Omron CX-Programmer project NewProject (CX-Programmer 9.74)

# PLC NewPLC1: CJ2M CPU32
I/O table (CPU CJ2M-CPU32): rack 0 slot 0 CJ1W-ID211; rack 0 slot 1 CJ1W-ID211; rack 0 slot 2 CJ1W-OD232; rack 0 slot 3 CJ1W-TC104; rack 0 slot 11 CJ2M-EIP21

## Data types
TYPE s_Steps : STRUCT
  f : INT;  (* Função *)
  p1 : INT;  (* Parametro 1 *)
  p2 : REAL;  (* Parametro 2 *)
END_STRUCT END_TYPE
TYPE s_Estado : STRUCT
  Ciclo : BOOL;  (* Em ciclo produtivo *)
  FimCiclo : BOOL;  (* Finalização ciclo *)
  Estado : BOOL;  (* Estado equipamento *)
  FimTratamento : BOOL;  (* Tratamento Finalizado *)
  OF_Carregada : BOOL;  (* Ordem carregada para máquina *)
  Avaria : BOOL;  (* Máquina em Avaria *)
  Com_OF : BOOL;  (* Máquina com OF carregada *)
  FalhaInjeProd : BOOL;  (* Falta de injeção de produto *)
  FalhaAquecim : BOOL;  (* Falha de aquecimento *)
  AvariaTermicos : BOOL;  (* Avaria de térmicos *)
  TratAbortado : BOOL;  (* Tratamento abortado pelo operador *)
  FalhaEnergia : BOOL;  (* Falha energia *)
  NivelProdBaixo : BOOL;  (* Nível produto químico no depósito baixo *)
  Manual : BOOL;  (* modo manual *)
  Emergencia : BOOL;  (* Paragem Emergência *)
END_STRUCT END_TYPE
TYPE s_of_pss : STRUCT  (* Passo individual do programa a executar *)
  f : INT;  (* Função *)
  p1 : INT;  (* Parametro 1 *)
  p2 : REAL;  (* Parametro 2 *)
  tt : REAL;  (* Totalizador *)
  uni : INT;  (* Unidade do totalizador *)
  rsv : INT Dimensions=[3];
END_STRUCT END_TYPE
TYPE s_pss_exe : STRUCT  (* Passo a executar *)
  pss : s_of_pss;  (* Passo actual a executar *)
  num_pss : INT;  (* Numero do passo actual *)
  ini : BOOL;  (* Inicio - Inicio do passo (Função faz inicializações necessárias) *)
  exe : BOOL;  (* Executar - Condição para funcionar (Função actua se valor igual a 1) *)
  fim : BOOL;  (* Fim - Terminado o passo (Função indica que terminou de executar) *)
  exc : BOOL;  (* Exclusivo - Condição para funções exclusivas (Função exclusiva coloca a 0 ao executar, impedindo que outras o façam) *)
END_STRUCT END_TYPE
TYPE s_trat : STRUCT
  Aspira : BOOL;
  Aquece : BOOL;
  Rotacao : BOOL;
  Injecao : BOOL;
  Ini : BOOL;
  Fim : BOOL;  (* Fim Passo *)
  CicloAtivo : BOOL;
  FimTratamento : BOOL;
END_STRUCT END_TYPE
TYPE s_of : STRUCT
  pss : s_of_pss Dimensions=[12];
END_STRUCT END_TYPE
TYPE s_of_net : STRUCT
  pss : s_Steps Dimensions=[12];
END_STRUCT END_TYPE

## Global symbols (name address type ; comment)
0.00 BOOL  ; Emerg:M1
0.00 BOOL  ; Emergency_M1
0.01 BOOL  ; Bt_start_M1
0.02 BOOL  ; Bt__Stop_M1
0.03 BOOL  ; selector de carga
0.04 BOOL  ; confirma carga
0.05 BOOL  ; Selector Descarga
0.06 BOOL  ; Confirma descarga
0.07 BOOL  ; Sns_flow_M1
0.08 BOOL  ; FC_PRT_M1
0.10 BOOL  ; conf rot M1
0.12 BOOL  ; Mgt_Resist_M1
0.13 BOOL  ; Emergencia
0.14 BOOL  ; bt_start
11.00 BOOL  ; Aux_ro_M1
12.00 BOOL  ; Aux_rot_M2
1.00 BOOL  ; Emerg:M2
1.01 BOOL  ; bt_inicio:M2
1.03 BOOL  ; selector de carga_M2
1.04 BOOL  ; conf carga_M2
1.05 BOOL  ; Sel Desc_M2
1.06 BOOL  ; Conf desc M2
1.07 BOOL  ; Sns_flow_M2
1.08 BOOL  ; FC_PRT_M2
1.10 BOOL  ; conf rot M2
1.12 BOOL  ; MGT_Resist_M2
1.13 BOOL  ; Cmt_Silo_1
1.14 BOOL  ; Cmt_Silo_2
2000 CHANNEL  ; Area_sp_Tc104_M1
2.00 BOOL  ; Girafa
2.01 BOOL  ; Tap_dist-DIR
2.02 BOOL  ; Out_Lig_desv1
2.03 BOOL  ; Out_Desl_desv1
2.04 BOOL  ; out_desv2
2.05 BOOL  ; Out_Desl_desv2
2.06 BOOL  ; Flap_Silo1
2.07 BOOL  ; Flap_Silo2
2.08 BOOL  ; Rotaçao_M1
2.09 BOOL  ; Resist_M1
2.10 BOOL  ; Valv_Aspira_M1
2.11 BOOL  ; Prt_Carga_M1
2.12 BOOL  ; Prt_Desc_M1
2.13 BOOL  ; lmp_auto_m1
2.14 BOOL  ; Lmp_Prt_carga_M1
2.15 BOOL  ; Lmp_Prt_Desc_M1
3.00 BOOL  ; Rotaçao_M2
3.01 BOOL  ; Resist_M2
3.02 BOOL  ; Valv_Aspira_M2
3.03 BOOL  ; Prt_Carga_M2
3.04 BOOL  ; Prt_Desc_M2
3.05 BOOL  ; lmp_auto_m2
3.06 BOOL  ; Lmp_Prt_carga_M2
3.07 BOOL  ; Lmp_Prt_Desc_M2
3.08 BOOL  ; lmp_Start_QE
3.09 BOOL  ; LMP_AVARIA_QE
3.10 BOOL  ; Led_Cmt_desv1
3.11 BOOL  ; Led_Cmt_desv2
3.12 BOOL  ; esquerda
3.13 BOOL  ; Vl_Inver_Tapete
3.14 BOOL  ; Baliza_M7
3.15 BOOL  ; Baliza_M8
C0001 BOOL  ; Cnt_CLC_1
C0002 BOOL  ; Cnt_CLC_2
C0003 BOOL  ; Cnt_CLC_3
C0004 BOOL  ; Cnt_CLC_4
C0005 BOOL  ; Cnt_CLC_5
C0011 BOOL  ; Cnt_CLC_1_M2
C0012 BOOL  ; Cnt_CLC_2_M2
C0013 BOOL  ; T_CLC_3_M2
C0014 BOOL  ; Cnt_CLC_4_M2
C0015 BOOL  ; Cnt_CLC_5_M2
D0 CHANNEL  ; Cntrl_Ns
D15 CHANNEL  ; Str_Msgs_M1
D16 CHANNEL  ; Pop_Inj_M2
D20 CHANNEL  ; T_CLC_1_M2
D21 CHANNEL  ; T_CLC_2
D22 CHANNEL  ; T_CLC_3
D23 CHANNEL  ; T_CLC_4
D24 CHANNEL  ; T_CLC_5
D25 CHANNEL  ; Str_Msgs_M1
D29 CHANNEL  ; Setp_temp_M1
D31 CHANNEL  ; T_CLC_2_M2
D32 CHANNEL  ; T_CLC_3_M2
D33 CHANNEL  ; T_CLC_4_M2
D34 CHANNEL  ; T_CLC_5_M2
D35 CHANNEL  ; Str_Msgs_M2
D38 CHANNEL  ; Area_sp_Tc104_M2
D39 CHANNEL  ; Setp_temp_M2
D5 CHANNEL  ; HMi_Notify
D6 CHANNEL  ; Pop_Inj_M1
D995 CHANNEL  ; Setp_Manual
D999 CHANNEL  ; Setp_Temp_NS
H0.00 BOOL  ; Auto_M1
H0.00 BOOL  ; Auto_M1
H0.08 BOOL  ; ALR ROTAÇAO
H0.09 BOOL  ; alarme_fluxo
H1 CHANNEL  ; passos prg M1
H10 CHANNEL  ; Ch_M2
H10.00 BOOL  ; Auto_M2
H10.08 BOOL  ; ALR ROT_M2
H10.09 BOOL  ; alr_fluxo_M2
H11 CHANNEL  ; passos prg M2
H11.00 BOOL  ; 1ªCICLO_M2
H11.01 BOOL  ; 2ªFNC_M2
H11.02 BOOL  ; 3ªCICLO_M2
H11.03 BOOL  ; 4ªFNC_M2
H11.04 BOOL  ; 5ªCICLO_M2
H11.05 BOOL  ; Fnc_Fim_M2
H12.00 BOOL  ; Fnc_1_dedust_M2
H12.01 BOOL  ; Fnc_1_Heat_M2
H12.03 BOOL  ; Fnc_INJ1_M2
H12.04 BOOL  ; Fnc_3_Dedust_M2
H12.05 BOOL  ; Fnc_3_Heat_M2
H12.07 BOOL  ; Fnc_INJ2_M2
H12.08 BOOL  ; Fnc_5_Dedust_M2
H12.09 BOOL  ; Fnc_5_Heat_M2
H13.04 BOOL  ; Mem Carga-M2
H13.05 BOOL  ; Mem_Desc-M2
H14.00 BOOL  ; MANUAL-M2
H14.01 BOOL  ; R ALARMES-M2
H14.02 BOOL  ; R INTERR AUT_M2
H1.00 BOOL  ; 1ªCICLO
H1.01 BOOL  ; 2ªFNC
H1.02 BOOL  ; 3ªCICLO
H1.03 BOOL  ; 4ªFNC
H1.04 BOOL  ; 5ªCICLO
H1.05 BOOL  ; Fnc_Fim_M1
H20.01 BOOL  ; Arranca Ciclo tapetes
H20.02 BOOL  ; Stop Ciclo Tapetes
H2.00 BOOL  ; Fnc_1_dedust
H2.01 BOOL  ; Fnc_1_Heat
H2.03 BOOL  ; Fnc_INJ1
H2.04 BOOL  ; Fnc_3_Dedust
H2.05 BOOL  ; Fnc_3_Heat
H2.07 BOOL  ; Fnc_INJ2
H2.08 BOOL  ; Fnc_5_Dedust
H2.09 BOOL  ; Fnc_5_Heat
H3.04 BOOL  ; Mem Carga-M1
H3.05 BOOL  ; Mem_Desc-M1
H4.00 BOOL  ; MANUAL-M1
H4.01 BOOL  ; R ALARMES-M1
H4.02 BOOL  ; R INTERR AUT_M1
T0005 BOOL  ; t_fim_M1
T0006 BOOL  ; t_fim_M2
T0008 BOOL  ; t_det_rotaçao_M1
T0009 BOOL  ; t-det-fluxo-M1
T0010 BOOL  ; Reset_M2
T0018 BOOL  ; t_det_rotaçao_M2
T0019 BOOL  ; t-det-fluxo-M2
T0021 BOOL  ; T_arranc_girafa
T0022 BOOL  ; Dlay_stop_Tap_distrib
T0023 BOOL  ; Dlay_stop_fch_valvs
T0024 BOOL  ; T_Desl desv1
T0025 BOOL  ; t_desl_Out_fch1
T0026 BOOL  ; T_Desl desv2
T0027 BOOL  ; t_desl_Out_fch2
T0028 BOOL  ; T_Liga_p_esq
T0029 BOOL  ; T_Abre_silo1
T0049 BOOL  ; T_Abre_silo2
T1002 BOOL  ; ~
W0.00 BOOL  ; tcl_giraf
W0.01 BOOL  ; tcl_tap_dist
W0.02 BOOL  ; tcl_On_Off_Desv1
W0.03 BOOL  ; Tcl_On_Off_Desv2
W0.03 BOOL  ; tcl_lig_desv2
W0.04 BOOL  ; Tcl_INJ1_M1
W0.05 BOOL  ; Tcl_INJ2_M1
W0.06 BOOL  ; Tcl_Raz_Silo1
W0.07 BOOL  ; cond_V1
W0.08 BOOL  ; Tcl_Start_M1
W0.09 BOOL  ; Tcl_Stop_M1
W0.10 BOOL  ; tcl_Rotaçao_M1
W0.11 BOOL  ; Tcl_Aquece_M1
W0.12 BOOL  ; Tcl_Aspira_M1
W0.13 BOOL  ; Tcl_Load_M1
W0.14 BOOL  ; tcl_unload_M1
W0.15 BOOL  ; Cmd_Start_Stop
W10.08 BOOL  ; Tcl_Start_M2
W1.01 BOOL  ; Tcl_Tap_ESQ
W1.04 BOOL  ; Tcl_INJ1_M2
W1.05 BOOL  ; Tcl_INJ2_M2
W1.06 BOOL  ; Tcl_Raz_Silo2
W1.07 BOOL  ; cond_V2
W1.08 BOOL  ; Tcl_Start_M2
W1.09 BOOL  ; Tcl_Stop_M2
W1.10 BOOL  ; tcl_Rotaçao_M2
W1.11 BOOL  ; Tcl_Aquece_M2
W1.12 BOOL  ; Tcl_Aspira_M2
W1.13 BOOL  ; Tcl_Load_M1
W1.14 BOOL  ; Tcl_desc_m2
W2 CHANNEL  ; Ch_Lmps_Fnc
W3 CHANNEL  ; Ch_Lmps_Fnc_M2
W4 CHANNEL  ; Ch_Lmps_Fnc_M2
M7 Maquina
M7_StepsCopy fb_CopySteps
M7_Strings fb_maquina_pss_2_str10_PT
M8 Maquina
M8_StepsCopy fb_CopySteps
M8_Strings fb_maquina_pss_2_str10_PT
OFF CF114 BOOL
ON CF113 BOOL  ; System Normally On Flag
Reset_M1 T0000 BOOL  ; Reset_M1
ResiveFromMaster _CPU011_ReceiveData
in_BtnStopM8 1.02 BOOL
tt _CPU011_ReceiveData

## Program NewProgram1 (cyclic task 0)
Local symbols
Comm_Completion_Ok W101.03 BOOL
Comm_Error W101.04 BOOL
M7_BatchReal E0_5100 STRUCT s_Steps
M7_Estado E0_5107 STRUCT s_Estado
M7_Manual H40.02 BOOL
M7_PassoAct D6400 STRUCT s_pss_exe
M7_Receita_Maq E0_5000 STRUCT s_of_net
M7_Receita_Maq_Ok E0_5048.00 BOOL
M7_TemperatOnline W103 INT
M7_Temperatura E0_5105 INT
M7_TranspDest E0_5106 UINT
M7_Trat D7000 STRUCT s_trat
M7_TratOffline H40.01 BOOL
M7_TratOnline H40.00 BOOL
M7_rcpMaquina D6000 STRUCT s_of
M7_rcpMaquina_Ok D6120.00 BOOL
M7_rcpMoega D6200 STRUCT s_of
M7_rcpMoega_Ok D6420.00 BOOL
M7eM8_CommBusy W101.02 BOOL
M8_BatchReal E0_5300 STRUCT s_Steps
M8_Estado E0_5307 STRUCT s_Estado
M8_Manual H41.02 BOOL
M8_PassoAct D6900 STRUCT s_pss_exe
M8_Receita_Maq E0_5200 STRUCT s_of_net
M8_Receita_Maq_Ok E0_5248.00 BOOL
M8_TemperatOnline W104 INT
M8_Temperatura E0_5305 INT
M8_TranspDest E0_5306 UINT
M8_Trat D7050 STRUCT s_trat
M8_TratOffline H41.01 BOOL
M8_TratOnline H41.00 BOOL
M8_rcpMaquina D6500 STRUCT s_of
M8_rcpMaquina_Ok D6620.00 BOOL
M8_rcpMoega D6700 STRUCT s_of
M8_rcpMoega_Ok D6920.00 BOOL
bit_M7AqueceOffline W100.08 BOOL
bit_M7AqueceOnline W100.07 BOOL
bit_M7Aquece_On W102.10 BOOL
bit_M7AspirOffline W100.06 BOOL
bit_M7AspirOnline W100.05 BOOL
bit_M7Carga W100.03 BOOL
bit_M7DCarga W100.04 BOOL
bit_M7InjOffline W100.12 BOOL
bit_M7InjOnline W100.11 BOOL
bit_M7TumbOffline W100.10 BOOL
bit_M7TumbOnline W100.09 BOOL
bit_M7_Avaria W102.07 BOOL
bit_M7_Disponivel W100.01 BOOL
bit_M7_FimDCarga W101.00 BOOL
bit_M7_Stop W102.08 BOOL
bit_M8AqueceOffline W102.02 BOOL
bit_M8AqueceOnline W102.01 BOOL
bit_M8Aquece_Ok W102.11 BOOL
bit_M8AspirOffline W102.00 BOOL
bit_M8AspirOnline W100.15 BOOL
bit_M8Carga W100.13 BOOL
bit_M8DCarga W100.14 BOOL
bit_M8InjOffline W102.06 BOOL
bit_M8InjOnline W102.05 BOOL
bit_M8TumbOffline W102.04 BOOL
bit_M8TumbOnline W102.03 BOOL
bit_M8_Disponivel W100.02 BOOL
bit_M8_FimDCarga W101.01 BOOL
bit_M8_Stop W102.09 BOOL
bt_stop_M2 1.02 BOOL  ; bt_stop_M2
f114 W100.00 BOOL
m7_str_act D5000 STRING[30]  ; String do passo actual
m7_str_pss0 D5030 STRING[30]  ; String do passo 0
m7_str_pss1 D5060 STRING[30]  ; String do passo 1
m7_str_pss10 D5330 STRING[30]  ; String do passo 10
m7_str_pss11 D5360 STRING[30]  ; String do passo 11
m7_str_pss2 D5090 STRING[30]  ; String do passo 2
m7_str_pss3 D5120 STRING[30]  ; String do passo 3
m7_str_pss4 D5150 STRING[30]  ; String do passo 4
m7_str_pss5 D5180 STRING[30]  ; String do passo 5
m7_str_pss6 D5210 STRING[30]  ; String do passo 6
m7_str_pss7 D5240 STRING[30]  ; String do passo 7
m7_str_pss8 D5270 STRING[30]  ; String do passo 8
m7_str_pss9 D5300 STRING[30]  ; String do passo 9
m8_str_act D5400 STRING[30]  ; String do passo actual
m8_str_pss0 D5430 STRING[30]  ; String do passo 0
m8_str_pss1 D5460 STRING[30]  ; String do passo 1
m8_str_pss10 D5730 STRING[30]  ; String do passo 10
m8_str_pss11 D5760 STRING[30]  ; String do passo 11
m8_str_pss2 D5490 STRING[30]  ; String do passo 2
m8_str_pss3 D5520 STRING[30]  ; String do passo 3
m8_str_pss4 D5550 STRING[30]  ; String do passo 4
m8_str_pss5 D5580 STRING[30]  ; String do passo 5
m8_str_pss6 D5610 STRING[30]  ; String do passo 6
m8_str_pss7 D5640 STRING[30]  ; String do passo 7
m8_str_pss8 D5670 STRING[30]  ; String do passo 8
m8_str_pss9 D5700 STRING[30]  ; String do passo 9
tcl_tap_dist_Esq W0.07 BOOL  ; Cond_V1
tmpTemper W500 INT

### Section MAQ7

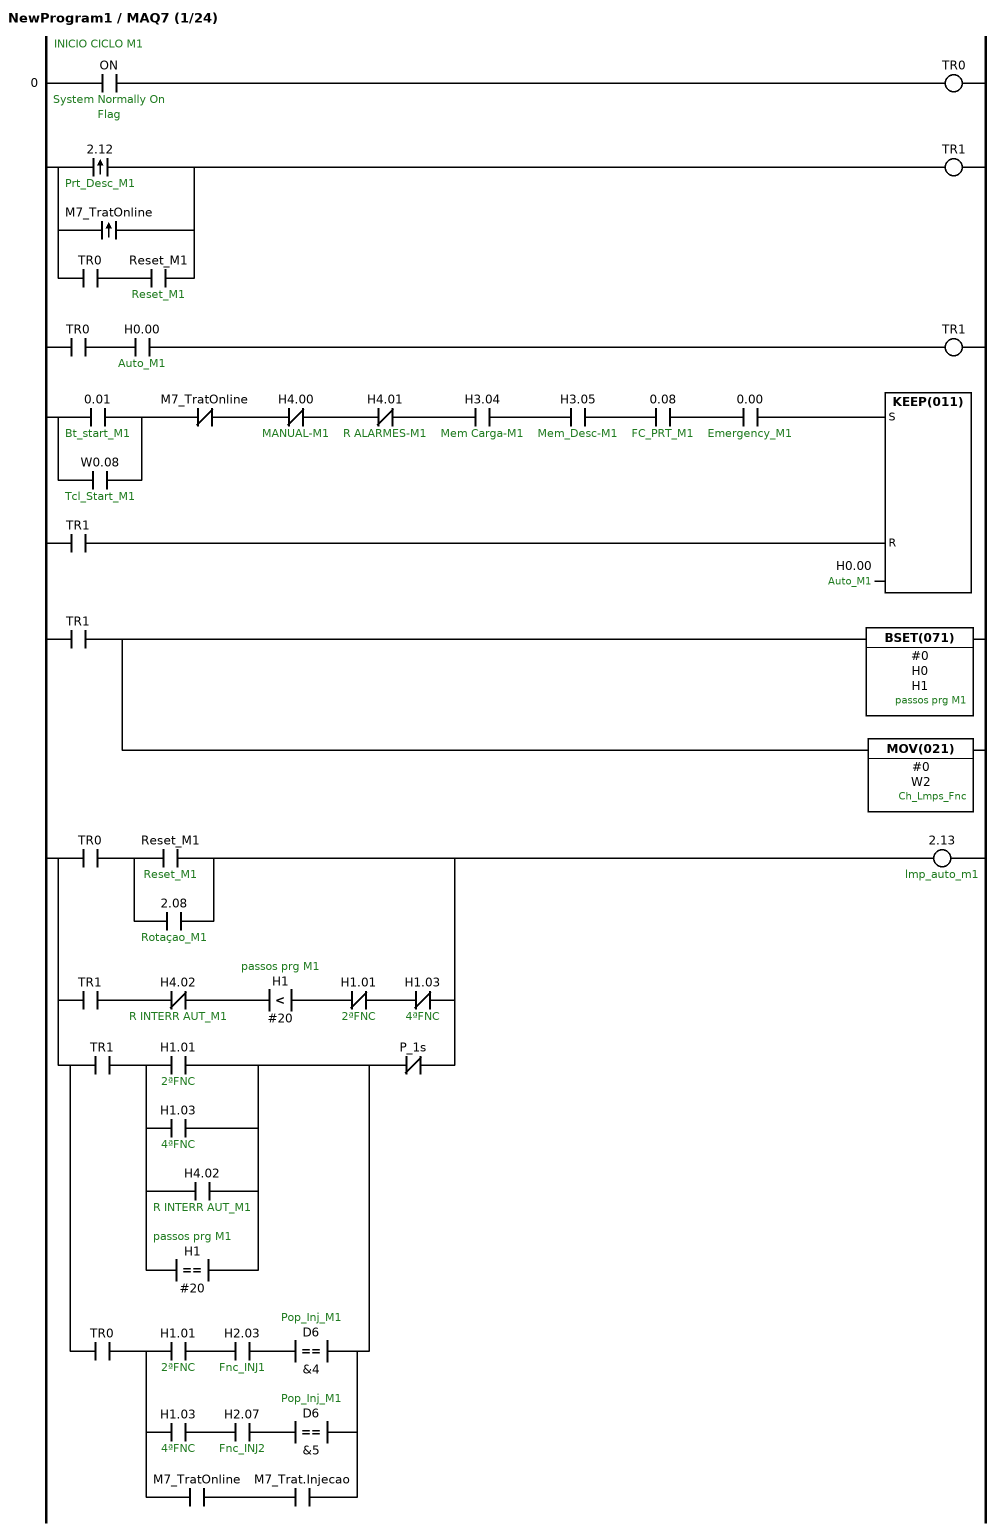
; rung 0: INICIO CICLO M1
LD 0.01  ; Bt_start_M1
OR W0.08  ; Tcl_Start_M1
ANDNOT M7_TratOnline
ANDNOT H4.00  ; MANUAL-M1
ANDNOT H4.01  ; R ALARMES-M1
AND H3.04  ; Mem Carga-M1
AND H3.05  ; Mem_Desc-M1
AND 0.08  ; FC_PRT_M1
AND 0.00  ; Emergency_M1
@LD 2.12  ; Prt_Desc_M1
@OR M7_TratOnline
LD ON  ; System Normally On Flag
OUT TR0
AND Reset_M1  ; Reset_M1
ORLD
OUT TR1
KEEP(011) H0.00  ; Auto_M1
LD TR1
BSET(071) #0 H0 H1  ; passos prg M1
MOV(021) #0 W2  ; Ch_Lmps_Fnc
LD TR0
LD Reset_M1  ; Reset_M1
OR 2.08  ; Rotaçao_M1
ANDLD
LD TR0
AND H0.00  ; Auto_M1
OUT TR1
ANDNOT H4.02  ; R INTERR AUT_M1
AND<(310) H1 #20  ; passos prg M1
ANDNOT H1.01  ; 2ªFNC
ANDNOT H1.03  ; 4ªFNC
ORLD
LD TR1
LD H1.01  ; 2ªFNC
OR H1.03  ; 4ªFNC
OR H4.02  ; R INTERR AUT_M1
OR=(300) H1 #20  ; passos prg M1
ANDLD
LD TR0
LD H1.01  ; 2ªFNC
AND H2.03  ; Fnc_INJ1
AND=(300) D6 &4  ; Pop_Inj_M1
LD H1.03  ; 4ªFNC
AND H2.07  ; Fnc_INJ2
AND=(300) D6 &5  ; Pop_Inj_M1
ORLD
LD M7_TratOnline
AND M7_Trat.Injecao
ORLD
ANDLD
ORLD
ANDNOT P_1s
ORLD
OUT 2.13  ; lmp_auto_m1

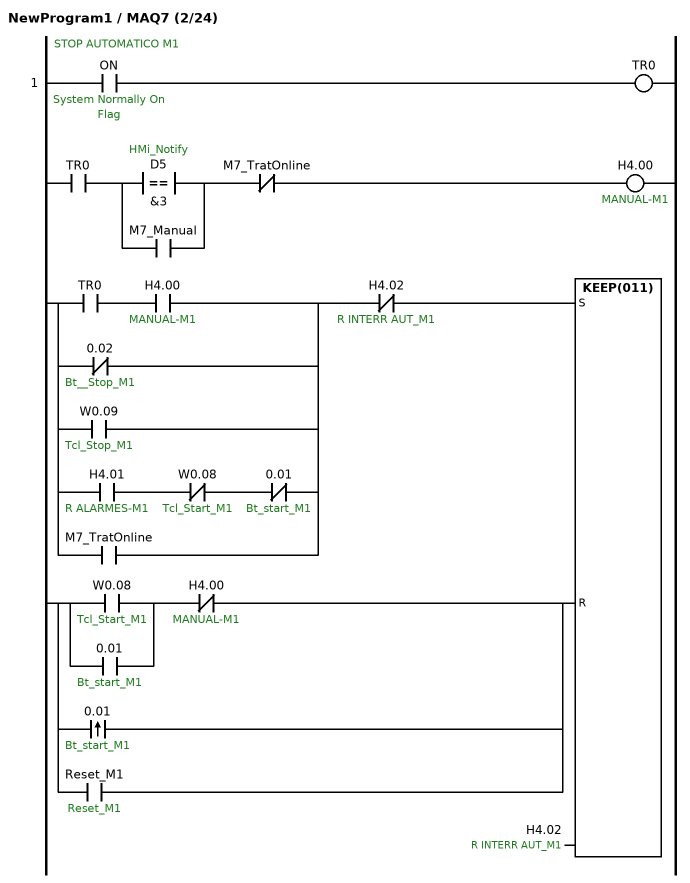
; rung 1: STOP AUTOMATICO M1
LD ON  ; System Normally On Flag
OUT TR0
LD=L(301) D5 &3  ; HMi_Notify
OR M7_Manual
ANDLD
ANDNOT M7_TratOnline
OUT H4.00  ; MANUAL-M1
LD TR0
AND H4.00  ; MANUAL-M1
LDNOT 0.02  ; Bt__Stop_M1
OR W0.09  ; Tcl_Stop_M1
LD H4.01  ; R ALARMES-M1
ANDNOT W0.08  ; Tcl_Start_M1
ANDNOT 0.01  ; Bt_start_M1
ORLD
OR M7_TratOnline
ORLD
ANDNOT H4.02  ; R INTERR AUT_M1
LD W0.08  ; Tcl_Start_M1
OR 0.01  ; Bt_start_M1
ANDNOT H4.00  ; MANUAL-M1
@OR 0.01  ; Bt_start_M1
OR Reset_M1  ; Reset_M1
KEEP(011) H4.02  ; R INTERR AUT_M1

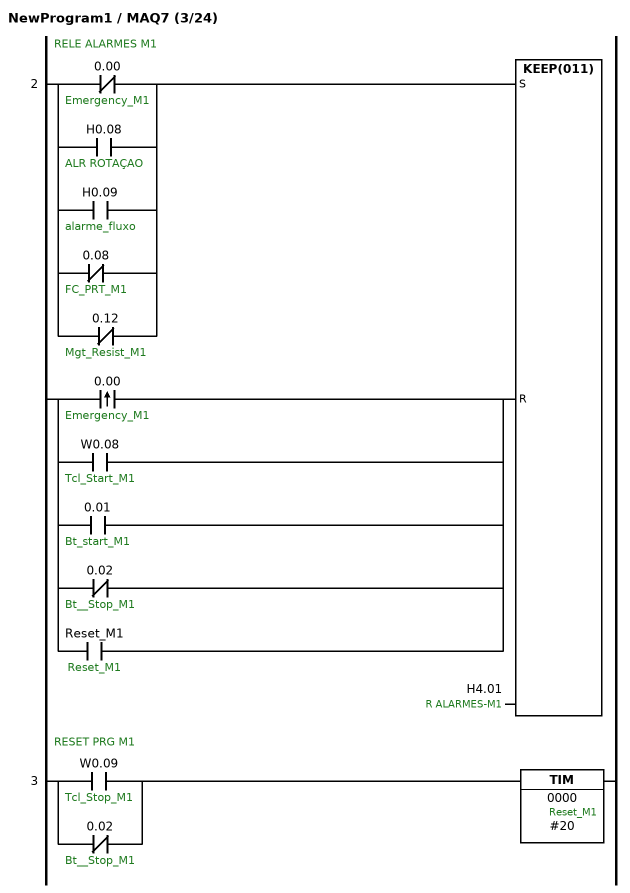
; rung 2: RELE ALARMES M1
LDNOT 0.00  ; Emergency_M1
OR H0.08  ; ALR ROTAÇAO
OR H0.09  ; alarme_fluxo
ORNOT 0.08  ; FC_PRT_M1
ORNOT 0.12  ; Mgt_Resist_M1
@LD 0.00  ; Emergency_M1
OR W0.08  ; Tcl_Start_M1
OR 0.01  ; Bt_start_M1
ORNOT 0.02  ; Bt__Stop_M1
OR Reset_M1  ; Reset_M1
KEEP(011) H4.01  ; R ALARMES-M1
; rung 3: RESET PRG M1
LD W0.09  ; Tcl_Stop_M1
ORNOT 0.02  ; Bt__Stop_M1
TIM 0000 #20  ; Reset_M1

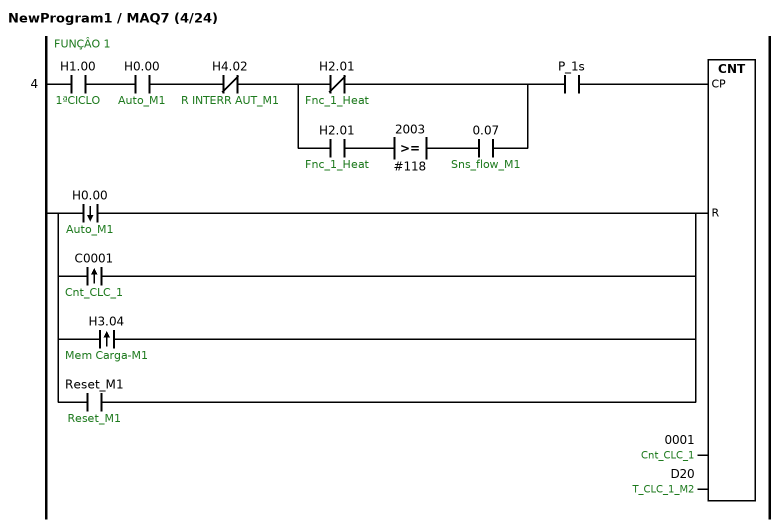
; rung 4: FUNÇÂO 1
LD H1.00  ; 1ªCICLO
AND H0.00  ; Auto_M1
ANDNOT H4.02  ; R INTERR AUT_M1
LDNOT H2.01  ; Fnc_1_Heat
LD H2.01  ; Fnc_1_Heat
AND>=(325) 2003 #118
AND 0.07  ; Sns_flow_M1
ORLD
ANDLD
AND P_1s
%LD H0.00  ; Auto_M1
@OR C0001  ; Cnt_CLC_1
@OR H3.04  ; Mem Carga-M1
OR Reset_M1  ; Reset_M1
CNT 0001 D20  ; T_CLC_1_M2, Cnt_CLC_1

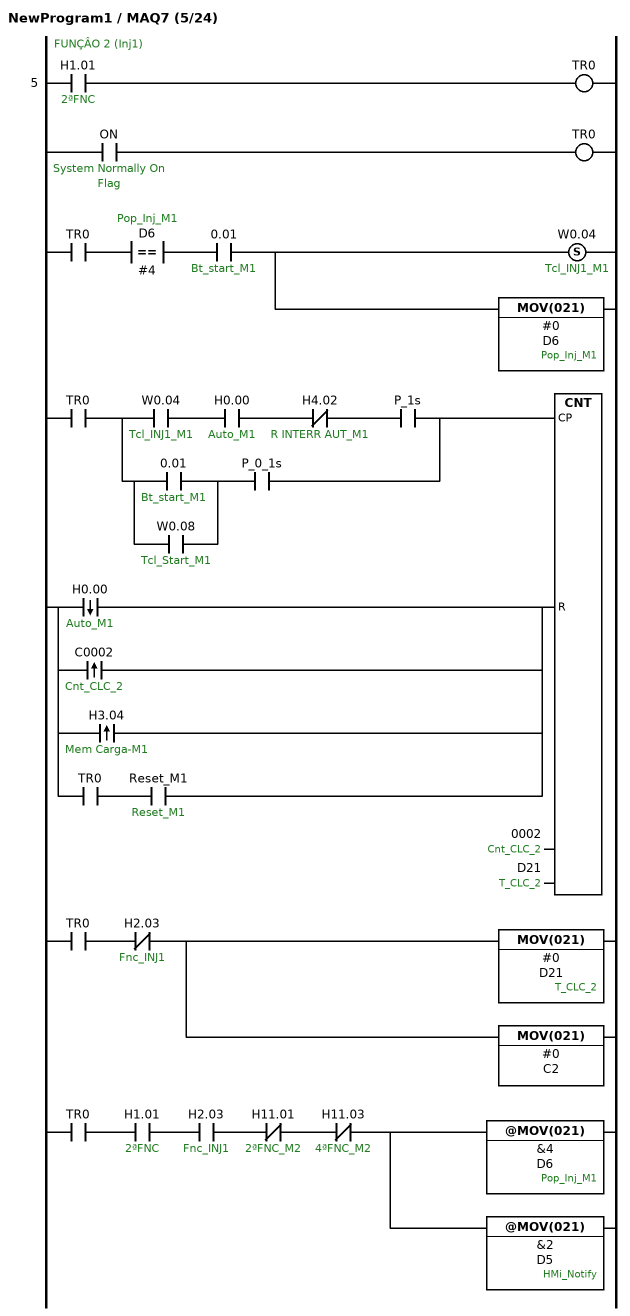
; rung 5: FUNÇÂO 2 (Inj1)
LD H1.01  ; 2ªFNC
OUT TR0
AND=(300) D6 #4  ; Pop_Inj_M1
AND 0.01  ; Bt_start_M1
SET W0.04  ; Tcl_INJ1_M1
MOV(021) #0 D6  ; Pop_Inj_M1
LD TR0
LD W0.04  ; Tcl_INJ1_M1
AND H0.00  ; Auto_M1
ANDNOT H4.02  ; R INTERR AUT_M1
AND P_1s
LD 0.01  ; Bt_start_M1
OR W0.08  ; Tcl_Start_M1
AND P_0_1s
ORLD
ANDLD
%LD H0.00  ; Auto_M1
@OR C0002  ; Cnt_CLC_2
@OR H3.04  ; Mem Carga-M1
LD ON  ; System Normally On Flag
OUT TR0
AND Reset_M1  ; Reset_M1
ORLD
CNT 0002 D21  ; T_CLC_2, Cnt_CLC_2
LD TR0
ANDNOT H2.03  ; Fnc_INJ1
MOV(021) #0 D21  ; T_CLC_2
MOV(021) #0 C2
LD TR0
AND H1.01  ; 2ªFNC
AND H2.03  ; Fnc_INJ1
ANDNOT H11.01  ; 2ªFNC_M2
ANDNOT H11.03  ; 4ªFNC_M2
@MOV(021) &4 D6  ; Pop_Inj_M1
@MOV(021) &2 D5  ; HMi_Notify

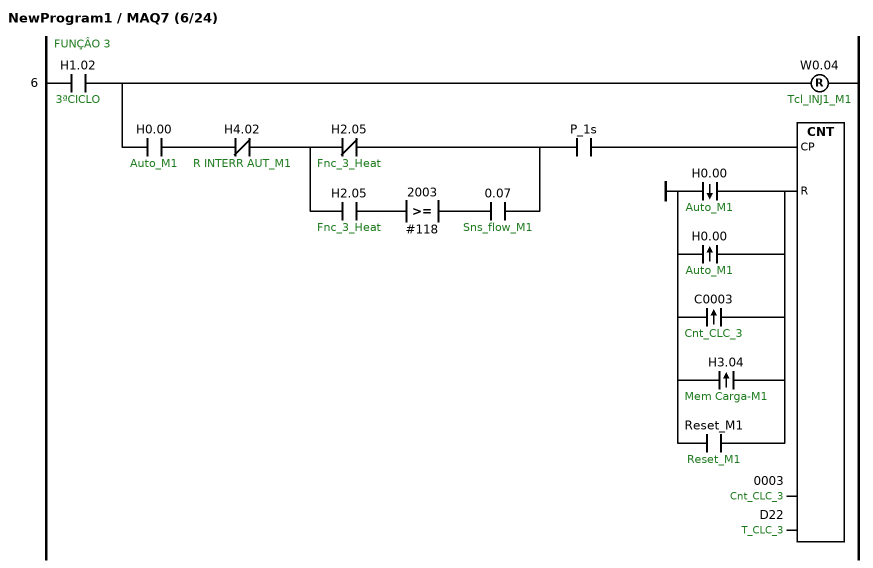
; rung 6: FUNÇÂO 3
LD H1.02  ; 3ªCICLO
RSET W0.04  ; Tcl_INJ1_M1
AND H0.00  ; Auto_M1
ANDNOT H4.02  ; R INTERR AUT_M1
LDNOT H2.05  ; Fnc_3_Heat
LD H2.05  ; Fnc_3_Heat
AND>=(325) 2003 #118
AND 0.07  ; Sns_flow_M1
ORLD
ANDLD
AND P_1s
%LD H0.00  ; Auto_M1
@OR H0.00  ; Auto_M1
@OR C0003  ; Cnt_CLC_3
@OR H3.04  ; Mem Carga-M1
OR Reset_M1  ; Reset_M1
CNT 0003 D22  ; T_CLC_3, Cnt_CLC_3

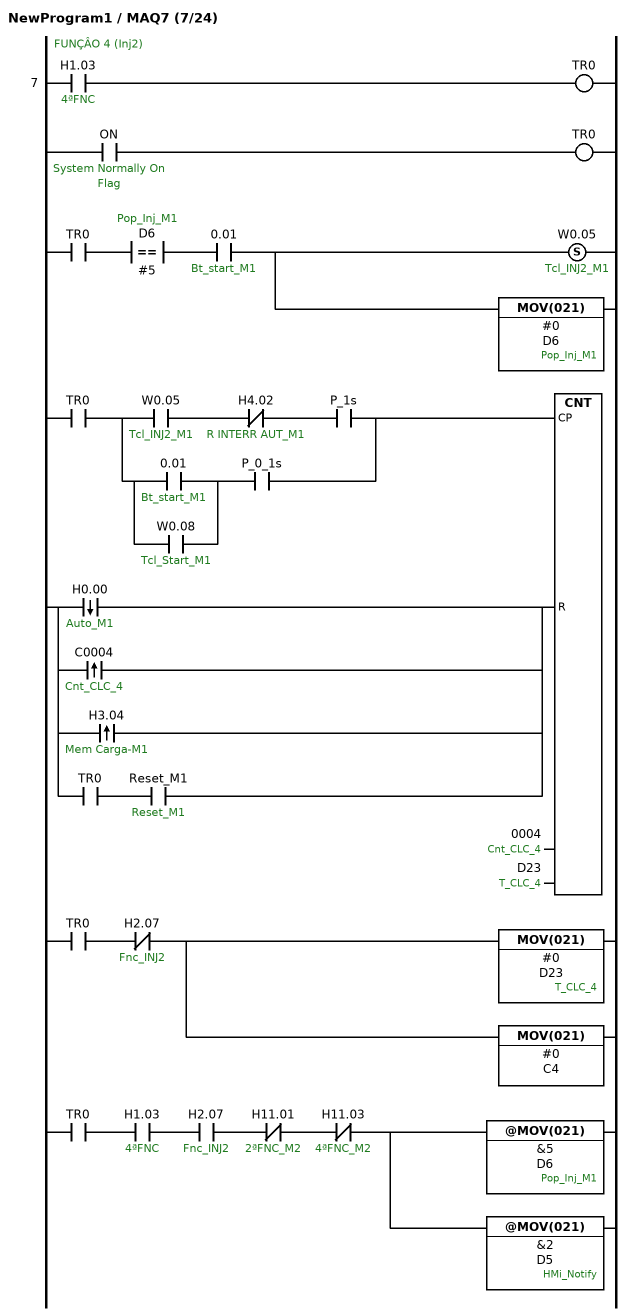
; rung 7: FUNÇÂO 4 (Inj2)
LD H1.03  ; 4ªFNC
OUT TR0
AND=(300) D6 #5  ; Pop_Inj_M1
AND 0.01  ; Bt_start_M1
SET W0.05  ; Tcl_INJ2_M1
MOV(021) #0 D6  ; Pop_Inj_M1
LD TR0
LD W0.05  ; Tcl_INJ2_M1
ANDNOT H4.02  ; R INTERR AUT_M1
AND P_1s
LD 0.01  ; Bt_start_M1
OR W0.08  ; Tcl_Start_M1
AND P_0_1s
ORLD
ANDLD
%LD H0.00  ; Auto_M1
@OR C0004  ; Cnt_CLC_4
@OR H3.04  ; Mem Carga-M1
LD ON  ; System Normally On Flag
OUT TR0
AND Reset_M1  ; Reset_M1
ORLD
CNT 0004 D23  ; T_CLC_4, Cnt_CLC_4
LD TR0
ANDNOT H2.07  ; Fnc_INJ2
MOV(021) #0 D23  ; T_CLC_4
MOV(021) #0 C4
LD TR0
AND H1.03  ; 4ªFNC
AND H2.07  ; Fnc_INJ2
ANDNOT H11.01  ; 2ªFNC_M2
ANDNOT H11.03  ; 4ªFNC_M2
@MOV(021) &5 D6  ; Pop_Inj_M1
@MOV(021) &2 D5  ; HMi_Notify

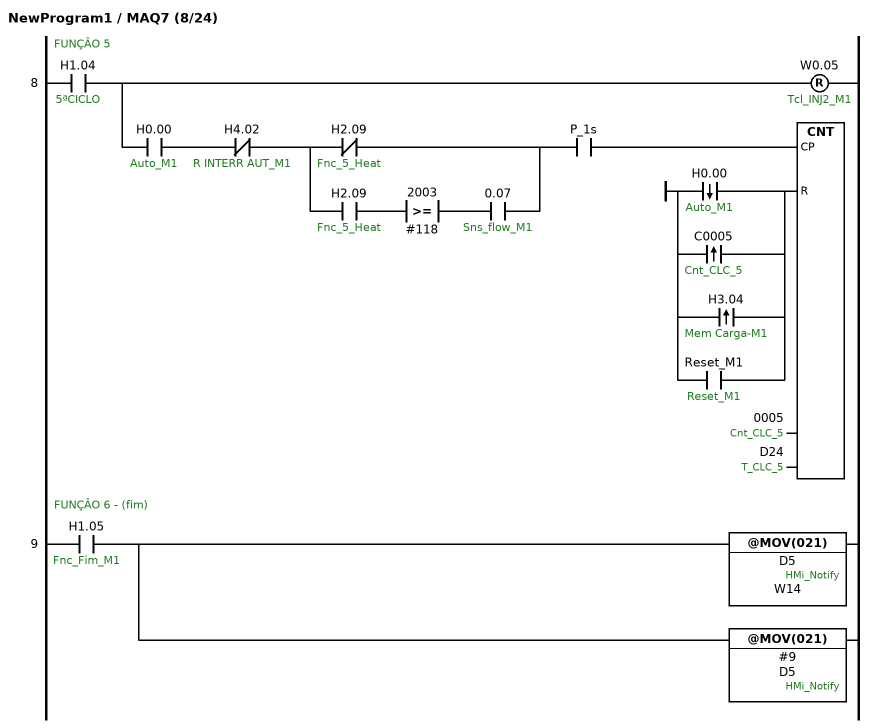
; rung 8: FUNÇÂO 5
LD H1.04  ; 5ªCICLO
RSET W0.05  ; Tcl_INJ2_M1
AND H0.00  ; Auto_M1
ANDNOT H4.02  ; R INTERR AUT_M1
LDNOT H2.09  ; Fnc_5_Heat
LD H2.09  ; Fnc_5_Heat
AND>=(325) 2003 #118
AND 0.07  ; Sns_flow_M1
ORLD
ANDLD
AND P_1s
%LD H0.00  ; Auto_M1
@OR C0005  ; Cnt_CLC_5
@OR H3.04  ; Mem Carga-M1
OR Reset_M1  ; Reset_M1
CNT 0005 D24  ; T_CLC_5, Cnt_CLC_5
; rung 9: FUNÇÂO 6 - (fim)
LD H1.05  ; Fnc_Fim_M1
@MOV(021) D5 W14  ; HMi_Notify
@MOV(021) #9 D5  ; HMi_Notify

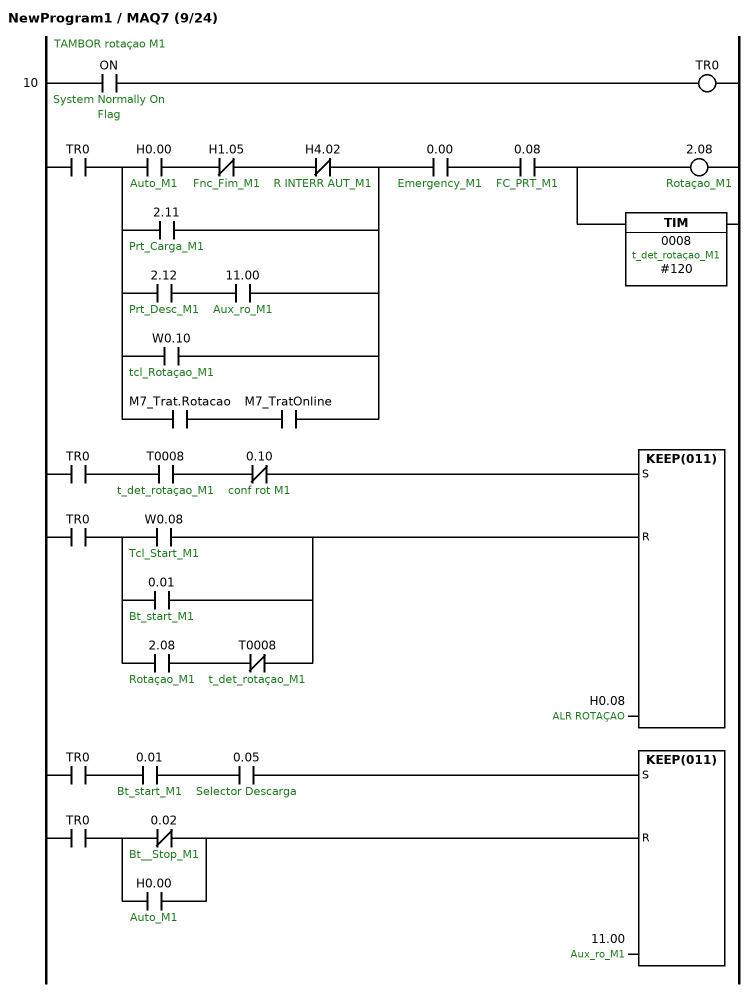
; rung 10: TAMBOR rotaçao M1
LD ON  ; System Normally On Flag
OUT TR0
LD H0.00  ; Auto_M1
ANDNOT H1.05  ; Fnc_Fim_M1
ANDNOT H4.02  ; R INTERR AUT_M1
OR 2.11  ; Prt_Carga_M1
LD 2.12  ; Prt_Desc_M1
AND 11.00  ; Aux_ro_M1
ORLD
OR W0.10  ; tcl_Rotaçao_M1
LD M7_Trat.Rotacao
AND M7_TratOnline
ORLD
ANDLD
AND 0.00  ; Emergency_M1
AND 0.08  ; FC_PRT_M1
OUT 2.08  ; Rotaçao_M1
TIM 0008 #120  ; t_det_rotaçao_M1
LD TR0
AND T0008  ; t_det_rotaçao_M1
ANDNOT 0.10  ; conf rot M1
LD TR0
LD W0.08  ; Tcl_Start_M1
OR 0.01  ; Bt_start_M1
LD 2.08  ; Rotaçao_M1
ANDNOT T0008  ; t_det_rotaçao_M1
ORLD
ANDLD
KEEP(011) H0.08  ; ALR ROTAÇAO
LD TR0
AND 0.01  ; Bt_start_M1
AND 0.05  ; Selector Descarga
LD TR0
LDNOT 0.02  ; Bt__Stop_M1
OR H0.00  ; Auto_M1
ANDLD
KEEP(011) 11.00  ; Aux_ro_M1

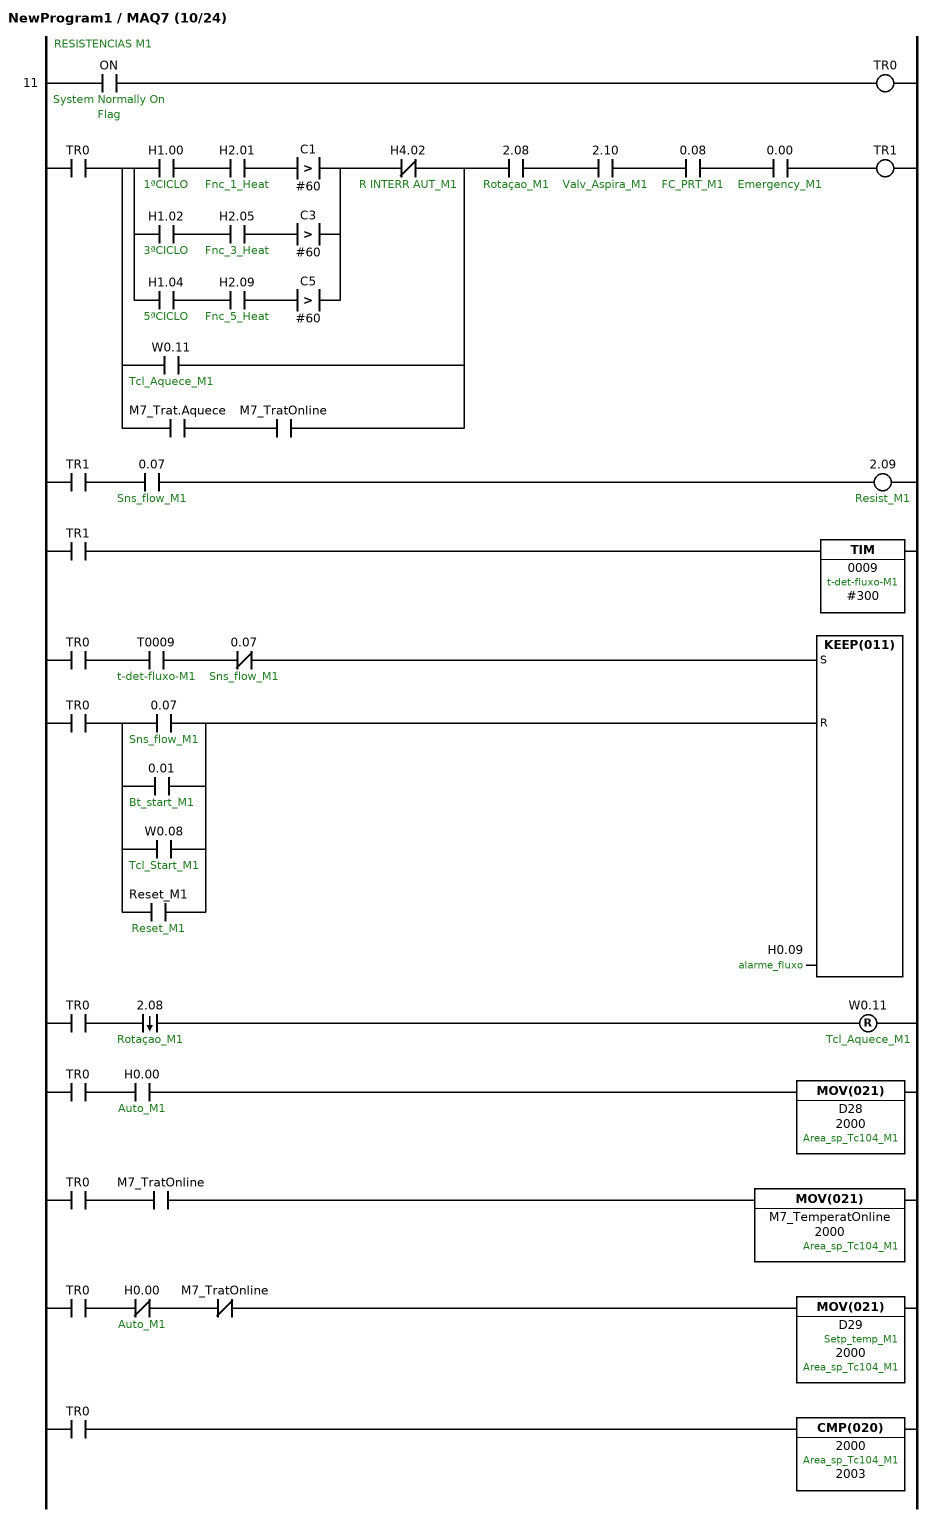
; rung 11: RESISTENCIAS M1
LD ON  ; System Normally On Flag
OUT TR0
LD H1.00  ; 1ªCICLO
AND H2.01  ; Fnc_1_Heat
AND>(320) C1 #60
LD H1.02  ; 3ªCICLO
AND H2.05  ; Fnc_3_Heat
AND>(320) C3 #60
ORLD
LD H1.04  ; 5ªCICLO
AND H2.09  ; Fnc_5_Heat
AND>(320) C5 #60
ORLD
ANDNOT H4.02  ; R INTERR AUT_M1
OR W0.11  ; Tcl_Aquece_M1
LD M7_Trat.Aquece
AND M7_TratOnline
ORLD
ANDLD
AND 2.08  ; Rotaçao_M1
AND 2.10  ; Valv_Aspira_M1
AND 0.08  ; FC_PRT_M1
AND 0.00  ; Emergency_M1
OUT TR1
AND 0.07  ; Sns_flow_M1
OUT 2.09  ; Resist_M1
LD TR1
TIM 0009 #300  ; t-det-fluxo-M1
LD TR0
AND T0009  ; t-det-fluxo-M1
ANDNOT 0.07  ; Sns_flow_M1
LD TR0
LD 0.07  ; Sns_flow_M1
OR 0.01  ; Bt_start_M1
OR W0.08  ; Tcl_Start_M1
OR Reset_M1  ; Reset_M1
ANDLD
KEEP(011) H0.09  ; alarme_fluxo
LD TR0
%AND 2.08  ; Rotaçao_M1
RSET W0.11  ; Tcl_Aquece_M1
LD TR0
AND H0.00  ; Auto_M1
MOV(021) D28 2000  ; Area_sp_Tc104_M1
LD TR0
AND M7_TratOnline
MOV(021) M7_TemperatOnline 2000  ; Area_sp_Tc104_M1
LD TR0
ANDNOT H0.00  ; Auto_M1
ANDNOT M7_TratOnline
MOV(021) D29 2000  ; Setp_temp_M1, Area_sp_Tc104_M1
LD TR0
CMP(020) 2000 2003  ; Area_sp_Tc104_M1

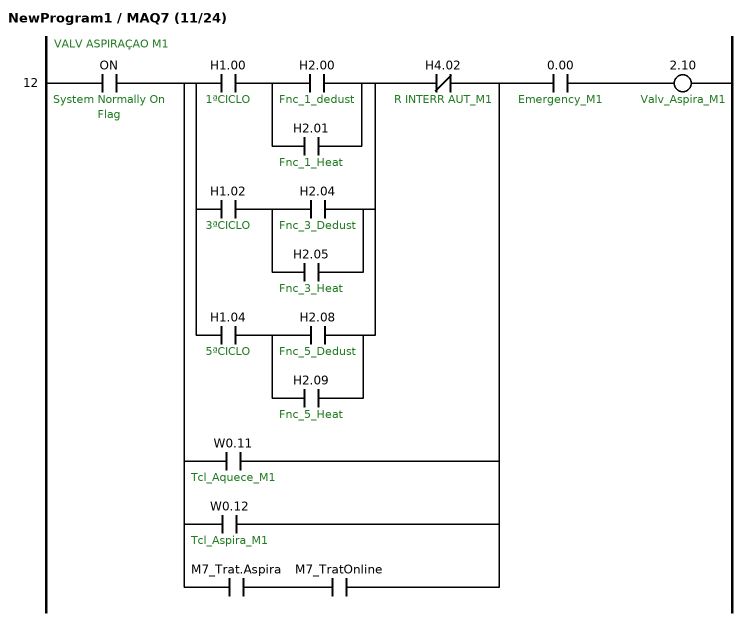
; rung 12: VALV ASPIRAÇAO M1
LD ON  ; System Normally On Flag
LD H1.00  ; 1ªCICLO
LD H2.00  ; Fnc_1_dedust
OR H2.01  ; Fnc_1_Heat
ANDLD
LD H1.02  ; 3ªCICLO
LD H2.04  ; Fnc_3_Dedust
OR H2.05  ; Fnc_3_Heat
ANDLD
ORLD
LD H1.04  ; 5ªCICLO
LD H2.08  ; Fnc_5_Dedust
OR H2.09  ; Fnc_5_Heat
ANDLD
ORLD
ANDNOT H4.02  ; R INTERR AUT_M1
OR W0.11  ; Tcl_Aquece_M1
OR W0.12  ; Tcl_Aspira_M1
LD M7_Trat.Aspira
AND M7_TratOnline
ORLD
ANDLD
AND 0.00  ; Emergency_M1
OUT 2.10  ; Valv_Aspira_M1

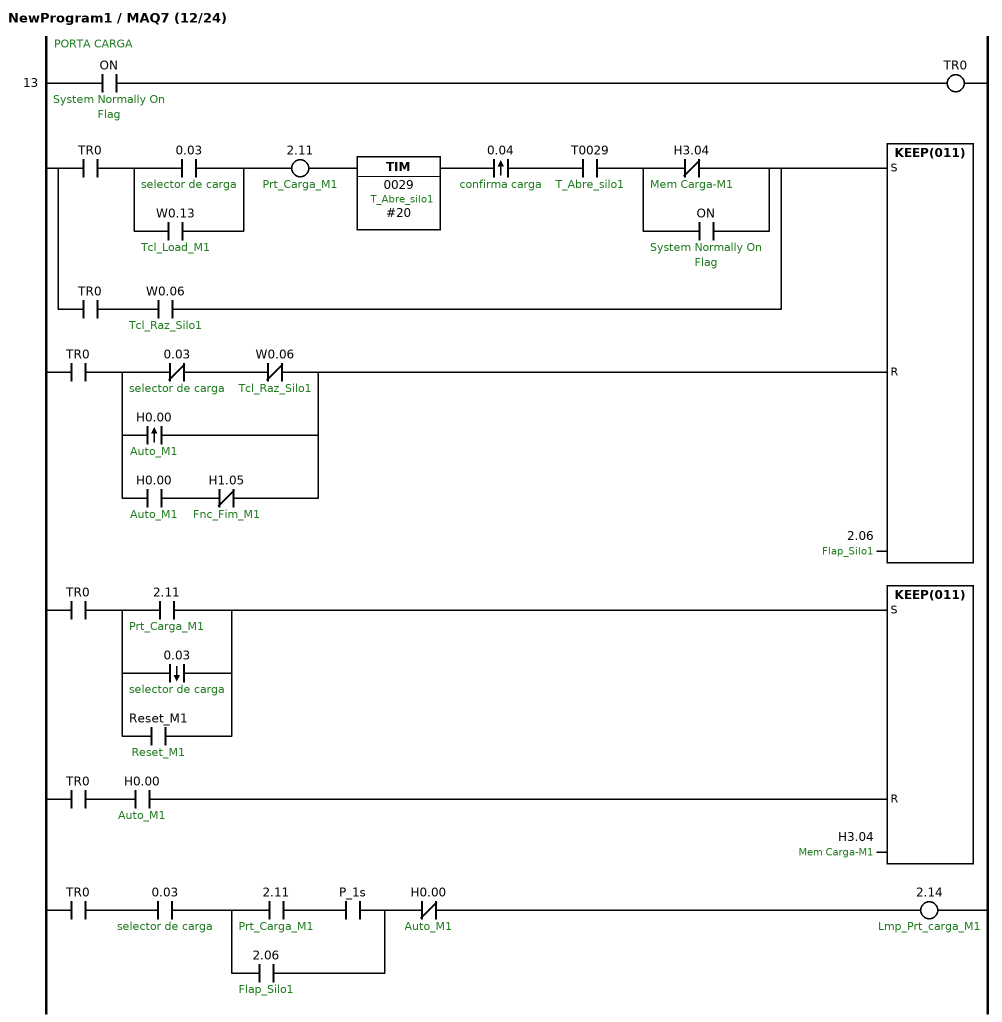
; rung 13: PORTA CARGA
LD ON  ; System Normally On Flag
OUT TR0
LD 0.03  ; selector de carga
OR W0.13  ; Tcl_Load_M1
ANDLD
OUT 2.11  ; Prt_Carga_M1
TIM 0029 #20  ; T_Abre_silo1
@AND 0.04  ; confirma carga
AND T0029  ; T_Abre_silo1
LDNOT H3.04  ; Mem Carga-M1
OR ON  ; System Normally On Flag
ANDLD
LD TR0
AND W0.06  ; Tcl_Raz_Silo1
ORLD
LD TR0
LDNOT 0.03  ; selector de carga
ANDNOT W0.06  ; Tcl_Raz_Silo1
@OR H0.00  ; Auto_M1
LD H0.00  ; Auto_M1
ANDNOT H1.05  ; Fnc_Fim_M1
ORLD
ANDLD
KEEP(011) 2.06  ; Flap_Silo1
LD TR0
LD 2.11  ; Prt_Carga_M1
%OR 0.03  ; selector de carga
OR Reset_M1  ; Reset_M1
ANDLD
LD TR0
AND H0.00  ; Auto_M1
KEEP(011) H3.04  ; Mem Carga-M1
LD TR0
AND 0.03  ; selector de carga
LD 2.11  ; Prt_Carga_M1
AND P_1s
OR 2.06  ; Flap_Silo1
ANDLD
ANDNOT H0.00  ; Auto_M1
OUT 2.14  ; Lmp_Prt_carga_M1

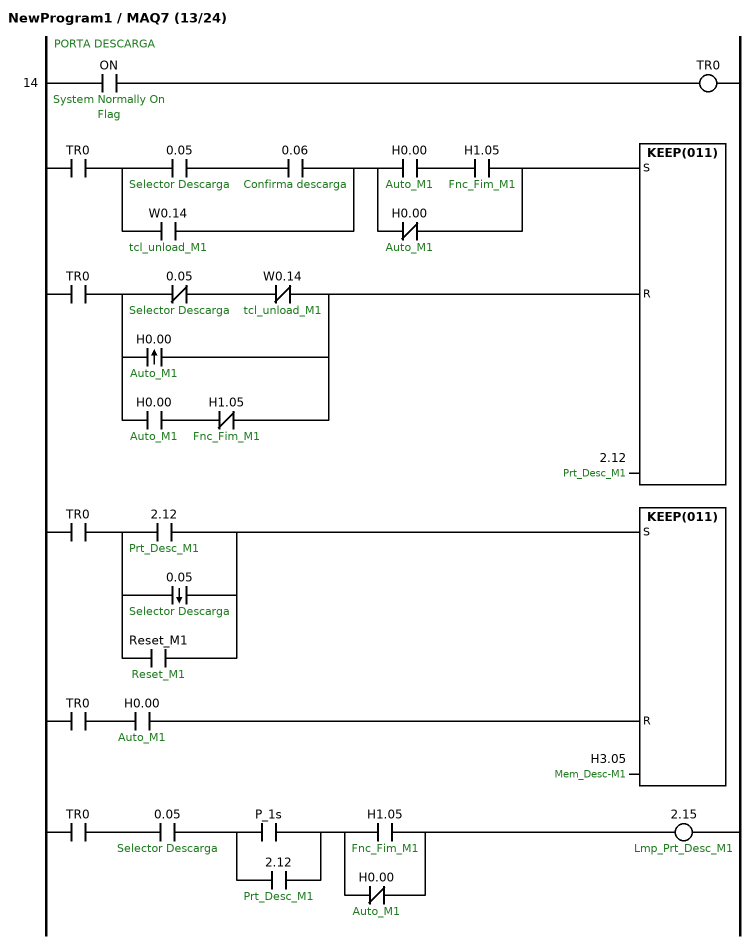
; rung 14: PORTA DESCARGA
LD ON  ; System Normally On Flag
OUT TR0
LD 0.05  ; Selector Descarga
AND 0.06  ; Confirma descarga
OR W0.14  ; tcl_unload_M1
ANDLD
LD H0.00  ; Auto_M1
AND H1.05  ; Fnc_Fim_M1
ORNOT H0.00  ; Auto_M1
ANDLD
LD TR0
LDNOT 0.05  ; Selector Descarga
ANDNOT W0.14  ; tcl_unload_M1
@OR H0.00  ; Auto_M1
LD H0.00  ; Auto_M1
ANDNOT H1.05  ; Fnc_Fim_M1
ORLD
ANDLD
KEEP(011) 2.12  ; Prt_Desc_M1
LD TR0
LD 2.12  ; Prt_Desc_M1
%OR 0.05  ; Selector Descarga
OR Reset_M1  ; Reset_M1
ANDLD
LD TR0
AND H0.00  ; Auto_M1
KEEP(011) H3.05  ; Mem_Desc-M1
LD TR0
AND 0.05  ; Selector Descarga
LD P_1s
OR 2.12  ; Prt_Desc_M1
ANDLD
LD H1.05  ; Fnc_Fim_M1
ORNOT H0.00  ; Auto_M1
ANDLD
OUT 2.15  ; Lmp_Prt_Desc_M1

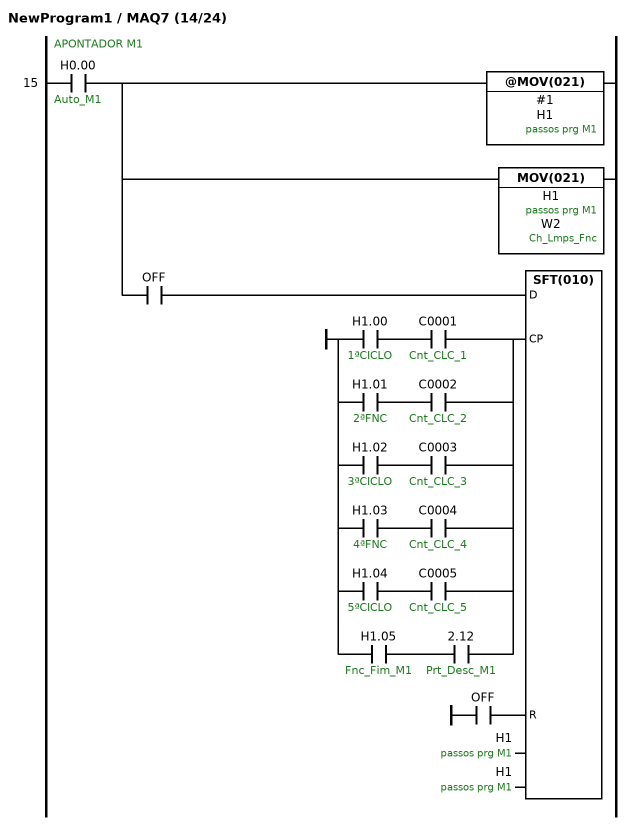
; rung 15: APONTADOR M1
LD H0.00  ; Auto_M1
@MOV(021) #1 H1  ; passos prg M1
MOV(021) H1 W2  ; passos prg M1, Ch_Lmps_Fnc
AND OFF
LD H1.00  ; 1ªCICLO
AND C0001  ; Cnt_CLC_1
LD H1.01  ; 2ªFNC
AND C0002  ; Cnt_CLC_2
ORLD
LD H1.02  ; 3ªCICLO
AND C0003  ; Cnt_CLC_3
ORLD
LD H1.03  ; 4ªFNC
AND C0004  ; Cnt_CLC_4
ORLD
LD H1.04  ; 5ªCICLO
AND C0005  ; Cnt_CLC_5
ORLD
LD H1.05  ; Fnc_Fim_M1
AND 2.12  ; Prt_Desc_M1
ORLD
LD OFF
SFT(010) H1 H1  ; passos prg M1

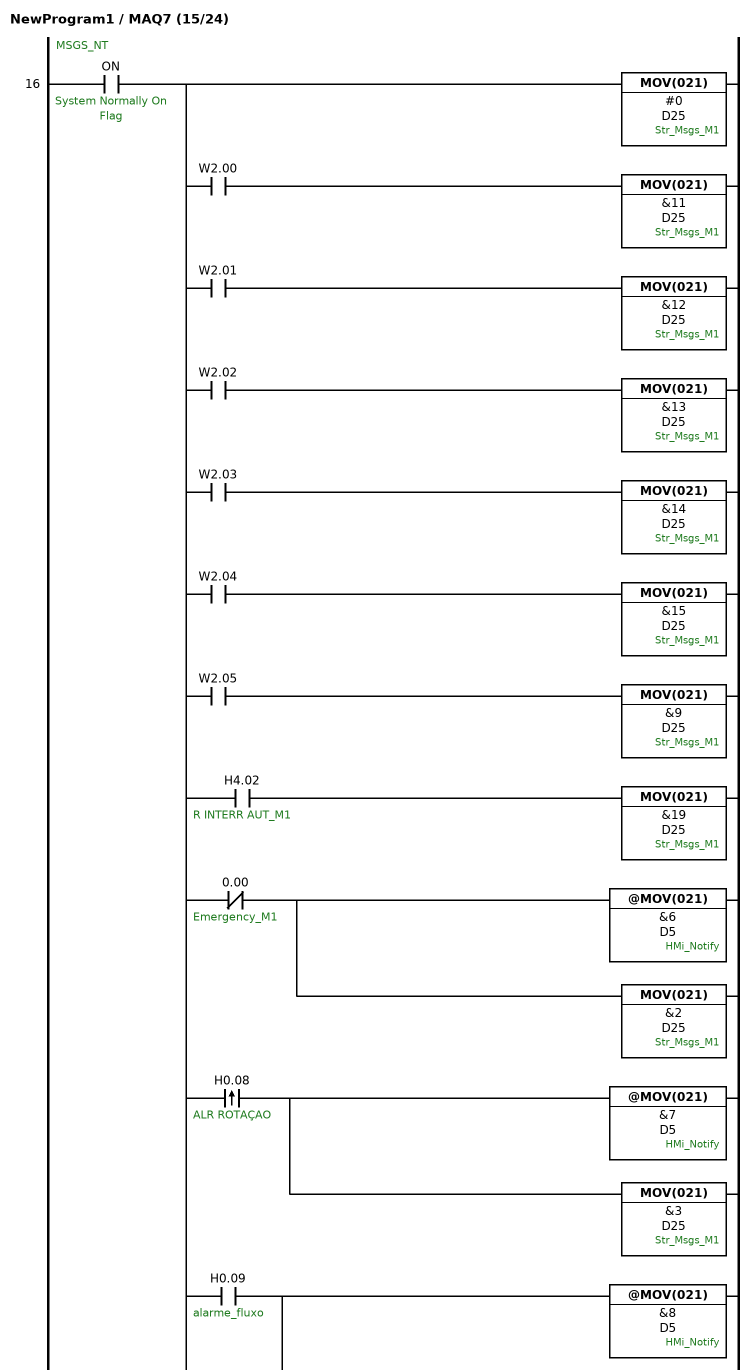

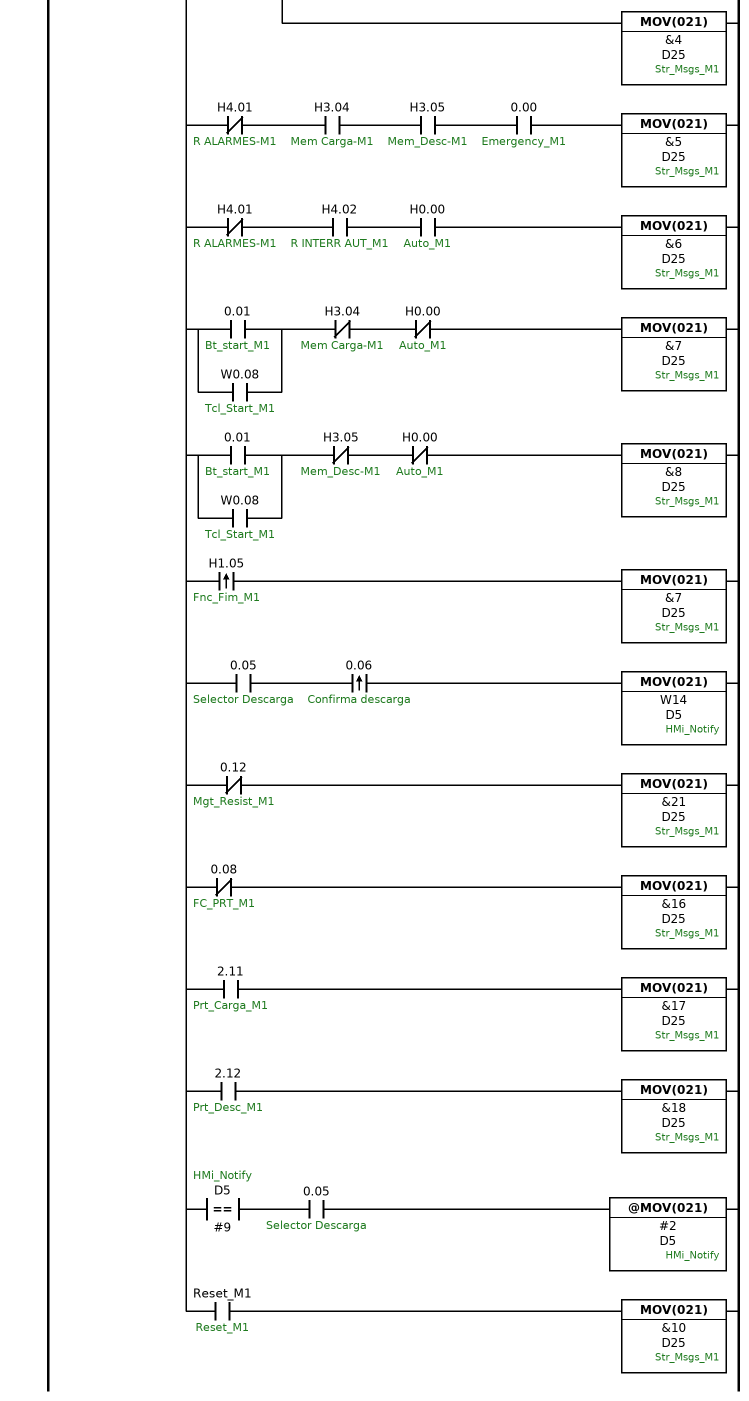
; rung 16: MSGS_NT
LD ON  ; System Normally On Flag
OUT TR0
MOV(021) #0 D25  ; Str_Msgs_M1
AND W2.00
MOV(021) &11 D25  ; Str_Msgs_M1
LD TR0
AND W2.01
MOV(021) &12 D25  ; Str_Msgs_M1
LD TR0
AND W2.02
MOV(021) &13 D25  ; Str_Msgs_M1
LD TR0
AND W2.03
MOV(021) &14 D25  ; Str_Msgs_M1
LD TR0
AND W2.04
MOV(021) &15 D25  ; Str_Msgs_M1
LD TR0
AND W2.05
MOV(021) &9 D25  ; Str_Msgs_M1
LD TR0
AND H4.02  ; R INTERR AUT_M1
MOV(021) &19 D25  ; Str_Msgs_M1
LD TR0
ANDNOT 0.00  ; Emergency_M1
@MOV(021) &6 D5  ; HMi_Notify
MOV(021) &2 D25  ; Str_Msgs_M1
LD TR0
@AND H0.08  ; ALR ROTAÇAO
@MOV(021) &7 D5  ; HMi_Notify
MOV(021) &3 D25  ; Str_Msgs_M1
LD TR0
AND H0.09  ; alarme_fluxo
@MOV(021) &8 D5  ; HMi_Notify
MOV(021) &4 D25  ; Str_Msgs_M1
LD TR0
ANDNOT H4.01  ; R ALARMES-M1
AND H3.04  ; Mem Carga-M1
AND H3.05  ; Mem_Desc-M1
AND 0.00  ; Emergency_M1
MOV(021) &5 D25  ; Str_Msgs_M1
LD TR0
ANDNOT H4.01  ; R ALARMES-M1
AND H4.02  ; R INTERR AUT_M1
AND H0.00  ; Auto_M1
MOV(021) &6 D25  ; Str_Msgs_M1
LD TR0
LD 0.01  ; Bt_start_M1
OR W0.08  ; Tcl_Start_M1
ANDLD
ANDNOT H3.04  ; Mem Carga-M1
ANDNOT H0.00  ; Auto_M1
MOV(021) &7 D25  ; Str_Msgs_M1
LD TR0
LD 0.01  ; Bt_start_M1
OR W0.08  ; Tcl_Start_M1
ANDLD
ANDNOT H3.05  ; Mem_Desc-M1
ANDNOT H0.00  ; Auto_M1
MOV(021) &8 D25  ; Str_Msgs_M1
LD TR0
@AND H1.05  ; Fnc_Fim_M1
MOV(021) &7 D25  ; Str_Msgs_M1
LD TR0
AND 0.05  ; Selector Descarga
@AND 0.06  ; Confirma descarga
MOV(021) W14 D5  ; HMi_Notify
LD TR0
ANDNOT 0.12  ; Mgt_Resist_M1
MOV(021) &21 D25  ; Str_Msgs_M1
LD TR0
ANDNOT 0.08  ; FC_PRT_M1
MOV(021) &16 D25  ; Str_Msgs_M1
LD TR0
AND 2.11  ; Prt_Carga_M1
MOV(021) &17 D25  ; Str_Msgs_M1
LD TR0
AND 2.12  ; Prt_Desc_M1
MOV(021) &18 D25  ; Str_Msgs_M1
LD TR0
AND=(300) D5 #9  ; HMi_Notify
AND 0.05  ; Selector Descarga
@MOV(021) #2 D5  ; HMi_Notify
LD TR0
AND Reset_M1  ; Reset_M1
MOV(021) &10 D25  ; Str_Msgs_M1

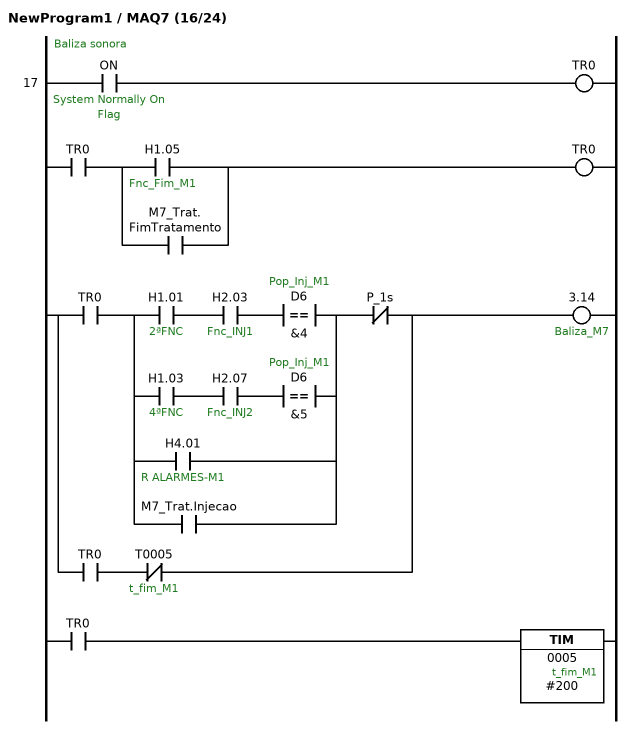
; rung 17: Baliza sonora
LD ON  ; System Normally On Flag
OUT TR0
LD H1.01  ; 2ªFNC
AND H2.03  ; Fnc_INJ1
AND=(300) D6 &4  ; Pop_Inj_M1
LD H1.03  ; 4ªFNC
AND H2.07  ; Fnc_INJ2
AND=(300) D6 &5  ; Pop_Inj_M1
ORLD
OR H4.01  ; R ALARMES-M1
OR M7_Trat.Injecao
ANDLD
ANDNOT P_1s
LD TR0
LD H1.05  ; Fnc_Fim_M1
OR M7_Trat.FimTratamento
ANDLD
OUT TR0
ANDNOT T0005  ; t_fim_M1
ORLD
OUT 3.14  ; Baliza_M7
LD TR0
TIM 0005 #200  ; t_fim_M1

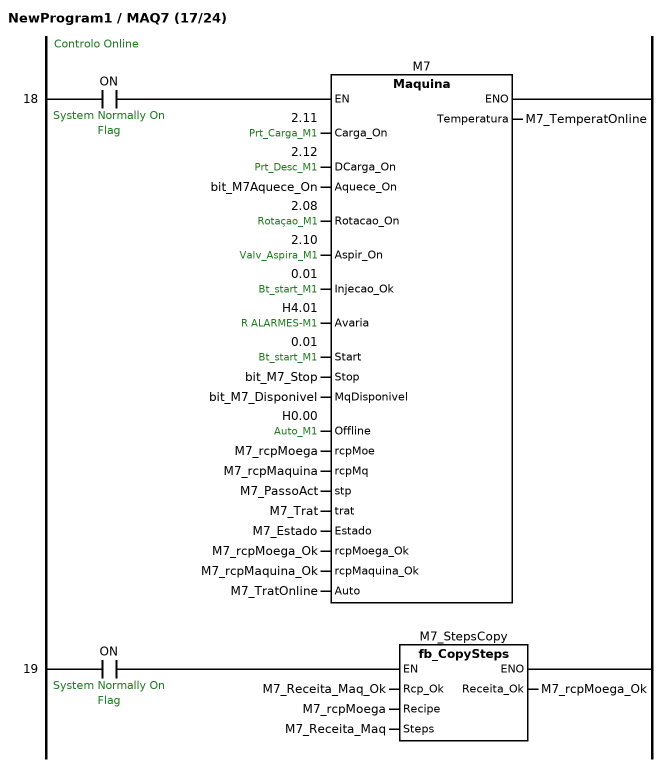
; rung 18: Controlo Online
LD ON  ; System Normally On Flag
CALL M7 : Maquina (Carga_On := 2.11, DCarga_On := 2.12, Aquece_On := bit_M7Aquece_On, Rotacao_On := 2.08, Aspir_On := 2.10, Injecao_Ok := 0.01, Avaria := H4.01, Start := 0.01, Stop := bit_M7_Stop, MqDisponivel := bit_M7_Disponivel, Offline := H0.00, rcpMoe := M7_rcpMoega, rcpMq := M7_rcpMaquina, stp := M7_PassoAct, trat := M7_Trat, Estado := M7_Estado, rcpMoega_Ok := M7_rcpMoega_Ok, rcpMaquina_Ok := M7_rcpMaquina_Ok, Auto := M7_TratOnline, Temperatura => M7_TemperatOnline)  ; Prt_Carga_M1, Prt_Desc_M1, Rotaçao_M1, Valv_Aspira_M1, Bt_start_M1, R ALARMES-M1, Auto_M1
; rung 19
LD ON  ; System Normally On Flag
CALL M7_StepsCopy : fb_CopySteps (Rcp_Ok := M7_Receita_Maq_Ok, Recipe := M7_rcpMoega, Steps := M7_Receita_Maq, Receita_Ok => M7_rcpMoega_Ok)

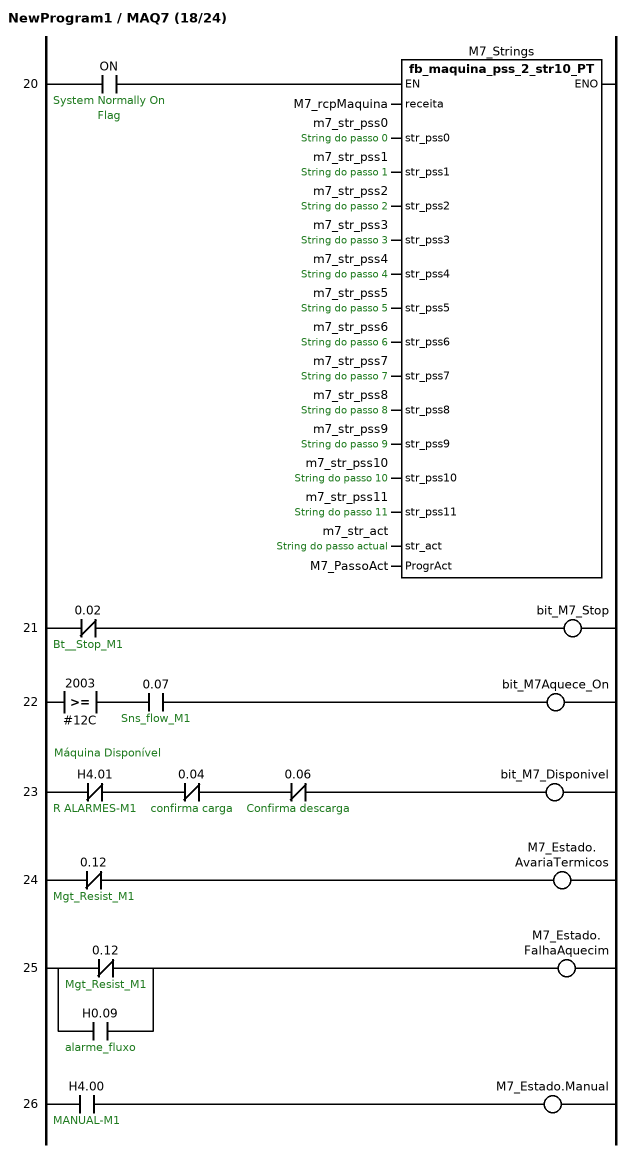
; rung 20
LD ON  ; System Normally On Flag
CALL M7_Strings : fb_maquina_pss_2_str10_PT (receita := M7_rcpMaquina, str_pss0 := m7_str_pss0, str_pss1 := m7_str_pss1, str_pss2 := m7_str_pss2, str_pss3 := m7_str_pss3, str_pss4 := m7_str_pss4, str_pss5 := m7_str_pss5, str_pss6 := m7_str_pss6, str_pss7 := m7_str_pss7, str_pss8 := m7_str_pss8, str_pss9 := m7_str_pss9, str_pss10 := m7_str_pss10, str_pss11 := m7_str_pss11, str_act := m7_str_act, ProgrAct := M7_PassoAct)  ; String do passo 0, String do passo 1, String do passo 2, String do passo 3, String do passo 4, String do passo 5, String do passo 6, String do passo 7, String do passo 8, String do passo 9, String do passo 10, String do passo 11, String do passo actual
; rung 21
LDNOT 0.02  ; Bt__Stop_M1
OUT bit_M7_Stop
; rung 22
LD>=(325) 2003 #12C
AND 0.07  ; Sns_flow_M1
OUT bit_M7Aquece_On
; rung 23: Máquina Disponível
LDNOT H4.01  ; R ALARMES-M1
ANDNOT 0.04  ; confirma carga
ANDNOT 0.06  ; Confirma descarga
OUT bit_M7_Disponivel
; rung 24
LDNOT 0.12  ; Mgt_Resist_M1
OUT M7_Estado.AvariaTermicos
; rung 25
LDNOT 0.12  ; Mgt_Resist_M1
OR H0.09  ; alarme_fluxo
OUT M7_Estado.FalhaAquecim
; rung 26
LD H4.00  ; MANUAL-M1
OUT M7_Estado.Manual

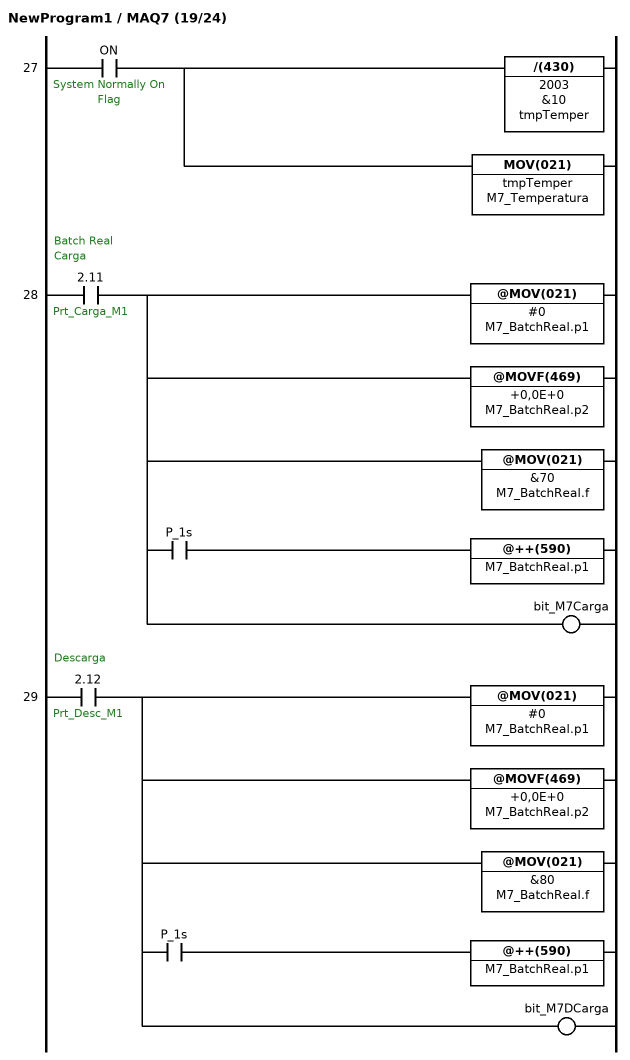
; rung 27
LD ON  ; System Normally On Flag
/(430) 2003 &10 tmpTemper
MOV(021) tmpTemper M7_Temperatura
; rung 28: Batch Real / Carga
LD 2.11  ; Prt_Carga_M1
OUT TR0
@MOV(021) #0 M7_BatchReal.p1
@MOVF(469) +0,0E+0 M7_BatchReal.p2
@MOV(021) &70 M7_BatchReal.f
AND P_1s
@++(590) M7_BatchReal.p1
LD TR0
OUT bit_M7Carga
; rung 29: Descarga
LD 2.12  ; Prt_Desc_M1
OUT TR0
@MOV(021) #0 M7_BatchReal.p1
@MOVF(469) +0,0E+0 M7_BatchReal.p2
@MOV(021) &80 M7_BatchReal.f
AND P_1s
@++(590) M7_BatchReal.p1
LD TR0
OUT bit_M7DCarga

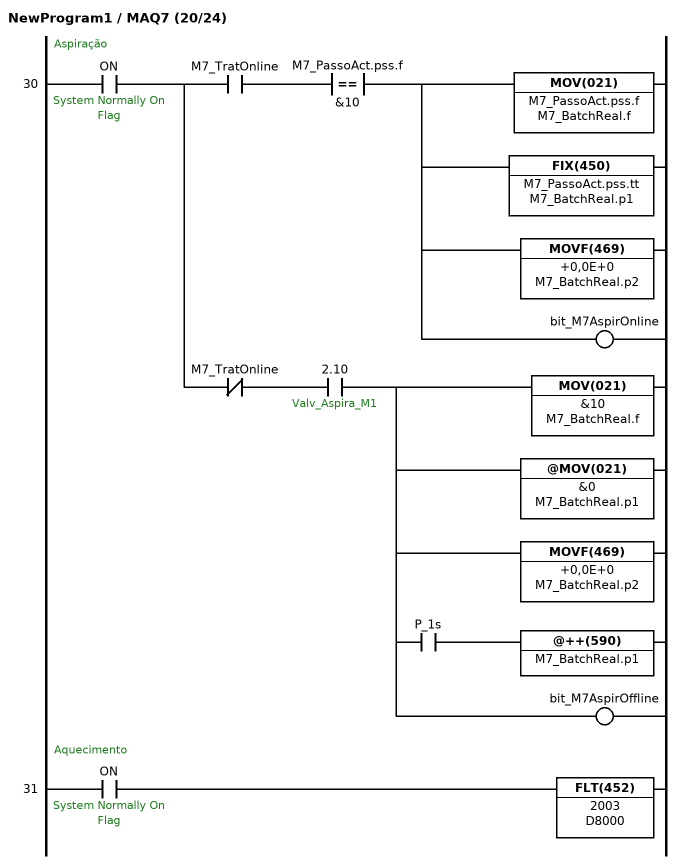
; rung 30: Aspiração
LD ON  ; System Normally On Flag
OUT TR0
AND M7_TratOnline
AND=(300) M7_PassoAct.pss.f &10
MOV(021) M7_PassoAct.pss.f M7_BatchReal.f
FIX(450) M7_PassoAct.pss.tt M7_BatchReal.p1
MOVF(469) +0,0E+0 M7_BatchReal.p2
OUT bit_M7AspirOnline
LD TR0
ANDNOT M7_TratOnline
AND 2.10  ; Valv_Aspira_M1
OUT TR0
MOV(021) &10 M7_BatchReal.f
@MOV(021) &0 M7_BatchReal.p1
MOVF(469) +0,0E+0 M7_BatchReal.p2
AND P_1s
@++(590) M7_BatchReal.p1
LD TR0
OUT bit_M7AspirOffline
; rung 31: Aquecimento
LD ON  ; System Normally On Flag
FLT(452) 2003 D8000

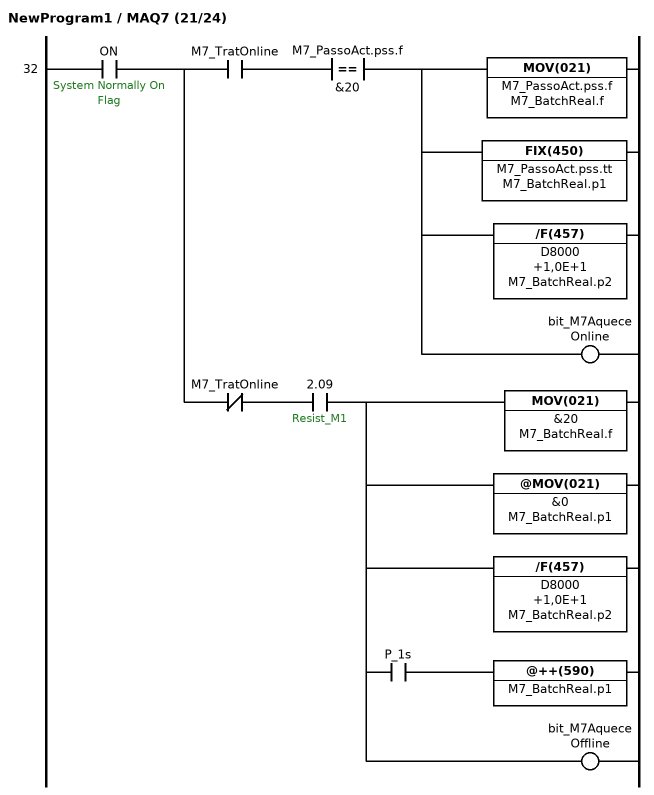
; rung 32
LD ON  ; System Normally On Flag
OUT TR0
AND M7_TratOnline
AND=(300) M7_PassoAct.pss.f &20
MOV(021) M7_PassoAct.pss.f M7_BatchReal.f
FIX(450) M7_PassoAct.pss.tt M7_BatchReal.p1
/F(457) D8000 +1,0E+1 M7_BatchReal.p2
OUT bit_M7AqueceOnline
LD TR0
ANDNOT M7_TratOnline
AND 2.09  ; Resist_M1
OUT TR0
MOV(021) &20 M7_BatchReal.f
@MOV(021) &0 M7_BatchReal.p1
/F(457) D8000 +1,0E+1 M7_BatchReal.p2
AND P_1s
@++(590) M7_BatchReal.p1
LD TR0
OUT bit_M7AqueceOffline

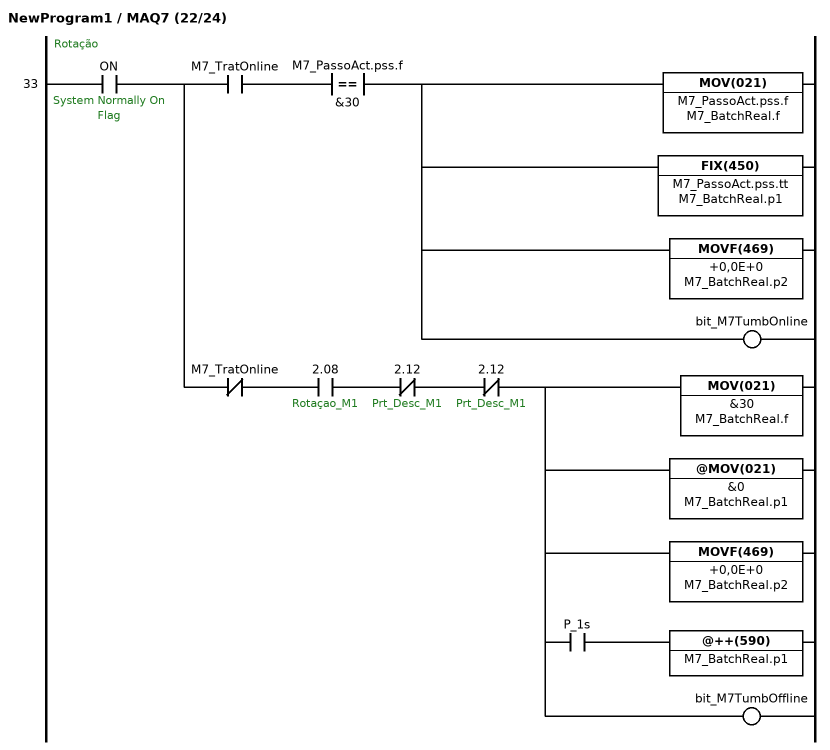
; rung 33: Rotação
LD ON  ; System Normally On Flag
OUT TR0
AND M7_TratOnline
AND=(300) M7_PassoAct.pss.f &30
MOV(021) M7_PassoAct.pss.f M7_BatchReal.f
FIX(450) M7_PassoAct.pss.tt M7_BatchReal.p1
MOVF(469) +0,0E+0 M7_BatchReal.p2
OUT bit_M7TumbOnline
LD TR0
ANDNOT M7_TratOnline
AND 2.08  ; Rotaçao_M1
ANDNOT 2.12  ; Prt_Desc_M1
ANDNOT 2.12  ; Prt_Desc_M1
OUT TR0
MOV(021) &30 M7_BatchReal.f
@MOV(021) &0 M7_BatchReal.p1
MOVF(469) +0,0E+0 M7_BatchReal.p2
AND P_1s
@++(590) M7_BatchReal.p1
LD TR0
OUT bit_M7TumbOffline

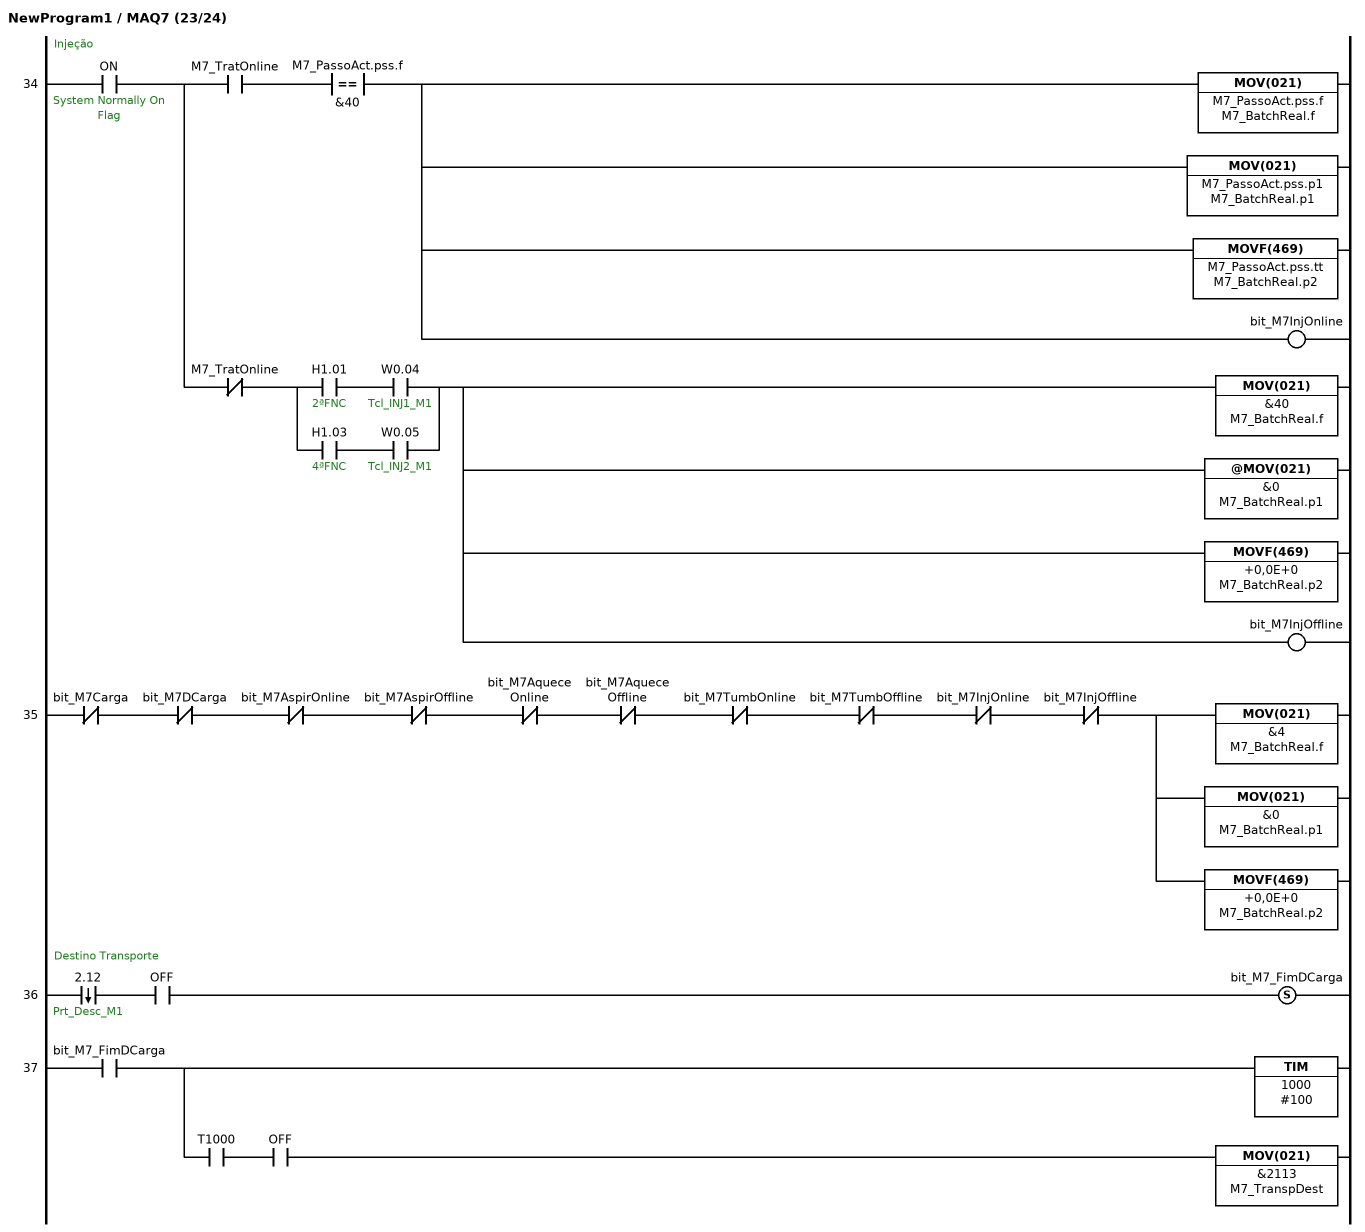
; rung 34: Injeção
LD ON  ; System Normally On Flag
OUT TR0
AND M7_TratOnline
AND=(300) M7_PassoAct.pss.f &40
MOV(021) M7_PassoAct.pss.f M7_BatchReal.f
MOV(021) M7_PassoAct.pss.p1 M7_BatchReal.p1
MOVF(469) M7_PassoAct.pss.tt M7_BatchReal.p2
OUT bit_M7InjOnline
LD TR0
ANDNOT M7_TratOnline
LD H1.01  ; 2ªFNC
AND W0.04  ; Tcl_INJ1_M1
LD H1.03  ; 4ªFNC
AND W0.05  ; Tcl_INJ2_M1
ORLD
ANDLD
MOV(021) &40 M7_BatchReal.f
@MOV(021) &0 M7_BatchReal.p1
MOVF(469) +0,0E+0 M7_BatchReal.p2
OUT bit_M7InjOffline
; rung 35
LDNOT bit_M7Carga
ANDNOT bit_M7DCarga
ANDNOT bit_M7AspirOnline
ANDNOT bit_M7AspirOffline
ANDNOT bit_M7AqueceOnline
ANDNOT bit_M7AqueceOffline
ANDNOT bit_M7TumbOnline
ANDNOT bit_M7TumbOffline
ANDNOT bit_M7InjOnline
ANDNOT bit_M7InjOffline
MOV(021) &4 M7_BatchReal.f
MOV(021) &0 M7_BatchReal.p1
MOVF(469) +0,0E+0 M7_BatchReal.p2
; rung 36: Destino Transporte
%LD 2.12  ; Prt_Desc_M1
AND OFF
SET bit_M7_FimDCarga
; rung 37
LD bit_M7_FimDCarga
TIM 1000 #100
AND T1000
AND OFF
MOV(021) &2113 M7_TranspDest

